// Mitsubishi GX Works2 project: B02_UDE 20260304_0   PLC: Q03UDE

PROGRAM 00  // Prog切替
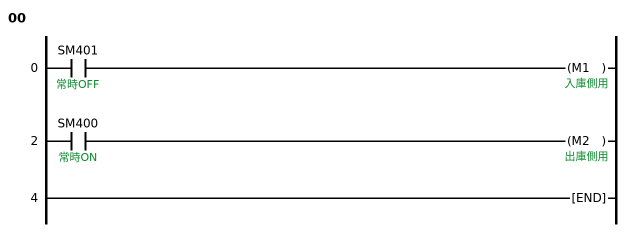
0     LD      SM401  ; 常時OFF
      OUT     M1  ; 入庫側用
2     LD      SM400  ; 常時ON
      OUT     M2  ; 出庫側用
4     END
END_PROGRAM

PROGRAM 01  // IO入力
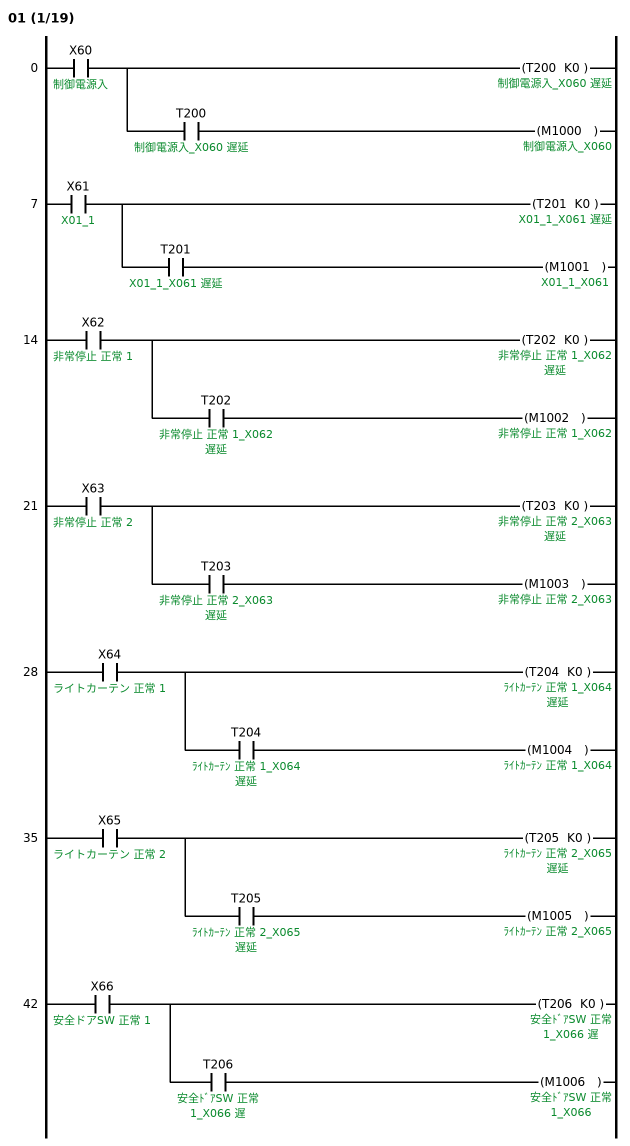
0     LD      X60  ; 制御電源入
      OUT     T200 K0  ; 制御電源入_X060 遅延
      AND     T200  ; 制御電源入_X060 遅延
      OUT     M1000  ; 制御電源入_X060
7     LD      X61  ; X01_1
      OUT     T201 K0  ; X01_1_X061 遅延
      AND     T201  ; X01_1_X061 遅延
      OUT     M1001  ; X01_1_X061
14    LD      X62  ; 非常停止 正常 1
      OUT     T202 K0  ; 非常停止 正常 1_X062 遅延
      AND     T202  ; 非常停止 正常 1_X062 遅延
      OUT     M1002  ; 非常停止 正常 1_X062
21    LD      X63  ; 非常停止 正常 2
      OUT     T203 K0  ; 非常停止 正常 2_X063 遅延
      AND     T203  ; 非常停止 正常 2_X063 遅延
      OUT     M1003  ; 非常停止 正常 2_X063
28    LD      X64  ; ライトカーテン 正常 1
      OUT     T204 K0  ; ﾗｲﾄｶｰﾃﾝ 正常 1_X064 遅延
      AND     T204  ; ﾗｲﾄｶｰﾃﾝ 正常 1_X064 遅延
      OUT     M1004  ; ﾗｲﾄｶｰﾃﾝ 正常 1_X064
35    LD      X65  ; ライトカーテン 正常 2
      OUT     T205 K0  ; ﾗｲﾄｶｰﾃﾝ 正常 2_X065 遅延
      AND     T205  ; ﾗｲﾄｶｰﾃﾝ 正常 2_X065 遅延
      OUT     M1005  ; ﾗｲﾄｶｰﾃﾝ 正常 2_X065
42    LD      X66  ; 安全ドアSW 正常 1
      OUT     T206 K0  ; 安全ﾄﾞｱSW 正常 1_X066 遅
      AND     T206  ; 安全ﾄﾞｱSW 正常 1_X066 遅
      OUT     M1006  ; 安全ﾄﾞｱSW 正常 1_X066
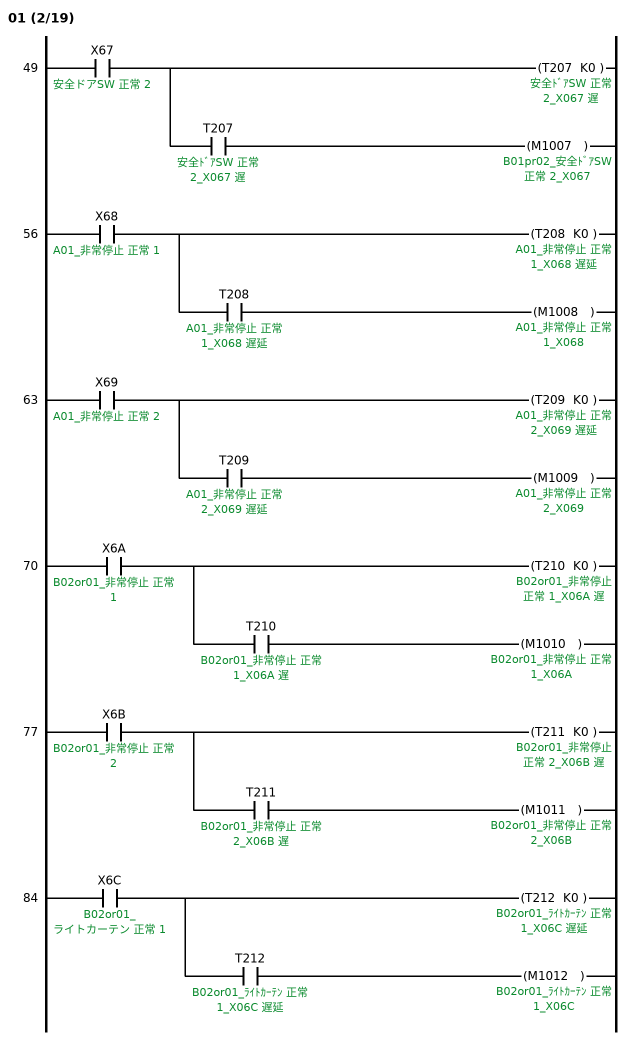
49    LD      X67  ; 安全ドアSW 正常 2
      OUT     T207 K0  ; 安全ﾄﾞｱSW 正常 2_X067 遅
      AND     T207  ; 安全ﾄﾞｱSW 正常 2_X067 遅
      OUT     M1007  ; B01pr02_安全ﾄﾞｱSW 正常 2_X067
56    LD      X68  ; A01_非常停止 正常 1
      OUT     T208 K0  ; A01_非常停止 正常 1_X068 遅延
      AND     T208  ; A01_非常停止 正常 1_X068 遅延
      OUT     M1008  ; A01_非常停止 正常 1_X068
63    LD      X69  ; A01_非常停止 正常 2
      OUT     T209 K0  ; A01_非常停止 正常 2_X069 遅延
      AND     T209  ; A01_非常停止 正常 2_X069 遅延
      OUT     M1009  ; A01_非常停止 正常 2_X069
70    LD      X6A  ; B02or01_非常停止 正常 1
      OUT     T210 K0  ; B02or01_非常停止 正常 1_X06A 遅
      AND     T210  ; B02or01_非常停止 正常 1_X06A 遅
      OUT     M1010  ; B02or01_非常停止 正常 1_X06A
77    LD      X6B  ; B02or01_非常停止 正常 2
      OUT     T211 K0  ; B02or01_非常停止 正常 2_X06B 遅
      AND     T211  ; B02or01_非常停止 正常 2_X06B 遅
      OUT     M1011  ; B02or01_非常停止 正常 2_X06B
84    LD      X6C  ; B02or01_ライトカーテン 正常 1
      OUT     T212 K0  ; B02or01_ﾗｲﾄｶｰﾃﾝ 正常 1_X06C 遅延
      AND     T212  ; B02or01_ﾗｲﾄｶｰﾃﾝ 正常 1_X06C 遅延
      OUT     M1012  ; B02or01_ﾗｲﾄｶｰﾃﾝ 正常 1_X06C
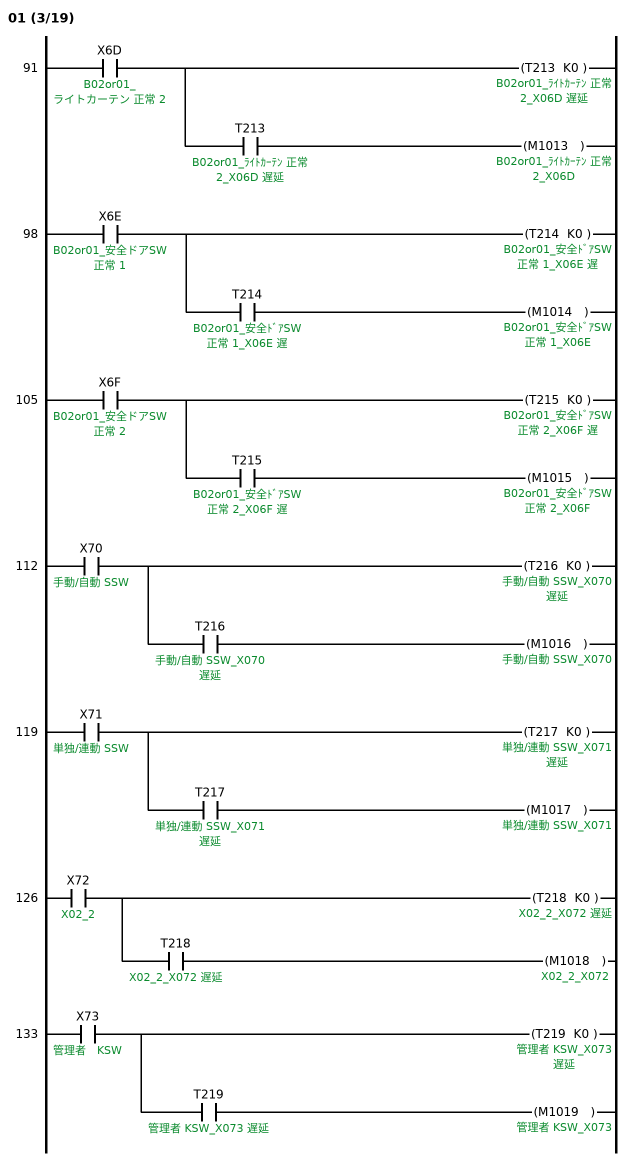
91    LD      X6D  ; B02or01_ライトカーテン 正常 2
      OUT     T213 K0  ; B02or01_ﾗｲﾄｶｰﾃﾝ 正常 2_X06D 遅延
      AND     T213  ; B02or01_ﾗｲﾄｶｰﾃﾝ 正常 2_X06D 遅延
      OUT     M1013  ; B02or01_ﾗｲﾄｶｰﾃﾝ 正常 2_X06D
98    LD      X6E  ; B02or01_安全ドアSW 正常 1
      OUT     T214 K0  ; B02or01_安全ﾄﾞｱSW 正常 1_X06E 遅
      AND     T214  ; B02or01_安全ﾄﾞｱSW 正常 1_X06E 遅
      OUT     M1014  ; B02or01_安全ﾄﾞｱSW 正常 1_X06E
105   LD      X6F  ; B02or01_安全ドアSW 正常 2
      OUT     T215 K0  ; B02or01_安全ﾄﾞｱSW 正常 2_X06F 遅
      AND     T215  ; B02or01_安全ﾄﾞｱSW 正常 2_X06F 遅
      OUT     M1015  ; B02or01_安全ﾄﾞｱSW 正常 2_X06F
112   LD      X70  ; 手動/自動 SSW
      OUT     T216 K0  ; 手動/自動 SSW_X070 遅延
      AND     T216  ; 手動/自動 SSW_X070 遅延
      OUT     M1016  ; 手動/自動 SSW_X070
119   LD      X71  ; 単独/連動 SSW
      OUT     T217 K0  ; 単独/連動 SSW_X071 遅延
      AND     T217  ; 単独/連動 SSW_X071 遅延
      OUT     M1017  ; 単独/連動 SSW_X071
126   LD      X72  ; X02_2
      OUT     T218 K0  ; X02_2_X072 遅延
      AND     T218  ; X02_2_X072 遅延
      OUT     M1018  ; X02_2_X072
133   LD      X73  ; 管理者　KSW
      OUT     T219 K0  ; 管理者 KSW_X073 遅延
      AND     T219  ; 管理者 KSW_X073 遅延
      OUT     M1019  ; 管理者 KSW_X073
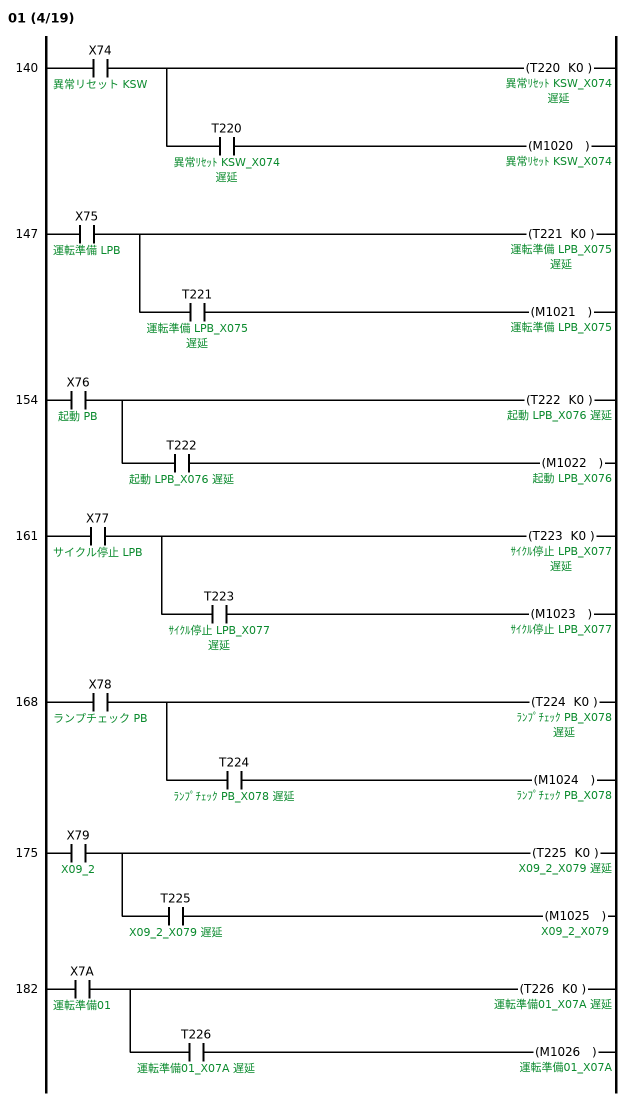
140   LD      X74  ; 異常リセット KSW
      OUT     T220 K0  ; 異常ﾘｾｯﾄ KSW_X074 遅延
      AND     T220  ; 異常ﾘｾｯﾄ KSW_X074 遅延
      OUT     M1020  ; 異常ﾘｾｯﾄ KSW_X074
147   LD      X75  ; 運転準備 LPB
      OUT     T221 K0  ; 運転準備 LPB_X075 遅延
      AND     T221  ; 運転準備 LPB_X075 遅延
      OUT     M1021  ; 運転準備 LPB_X075
154   LD      X76  ; 起動 PB
      OUT     T222 K0  ; 起動 LPB_X076 遅延
      AND     T222  ; 起動 LPB_X076 遅延
      OUT     M1022  ; 起動 LPB_X076
161   LD      X77  ; サイクル停止 LPB
      OUT     T223 K0  ; ｻｲｸﾙ停止 LPB_X077 遅延
      AND     T223  ; ｻｲｸﾙ停止 LPB_X077 遅延
      OUT     M1023  ; ｻｲｸﾙ停止 LPB_X077
168   LD      X78  ; ランプチェック PB
      OUT     T224 K0  ; ﾗﾝﾌﾟﾁｪｯｸ PB_X078 遅延
      AND     T224  ; ﾗﾝﾌﾟﾁｪｯｸ PB_X078 遅延
      OUT     M1024  ; ﾗﾝﾌﾟﾁｪｯｸ PB_X078
175   LD      X79  ; X09_2
      OUT     T225 K0  ; X09_2_X079 遅延
      AND     T225  ; X09_2_X079 遅延
      OUT     M1025  ; X09_2_X079
182   LD      X7A  ; 運転準備01
      OUT     T226 K0  ; 運転準備01_X07A 遅延
      AND     T226  ; 運転準備01_X07A 遅延
      OUT     M1026  ; 運転準備01_X07A
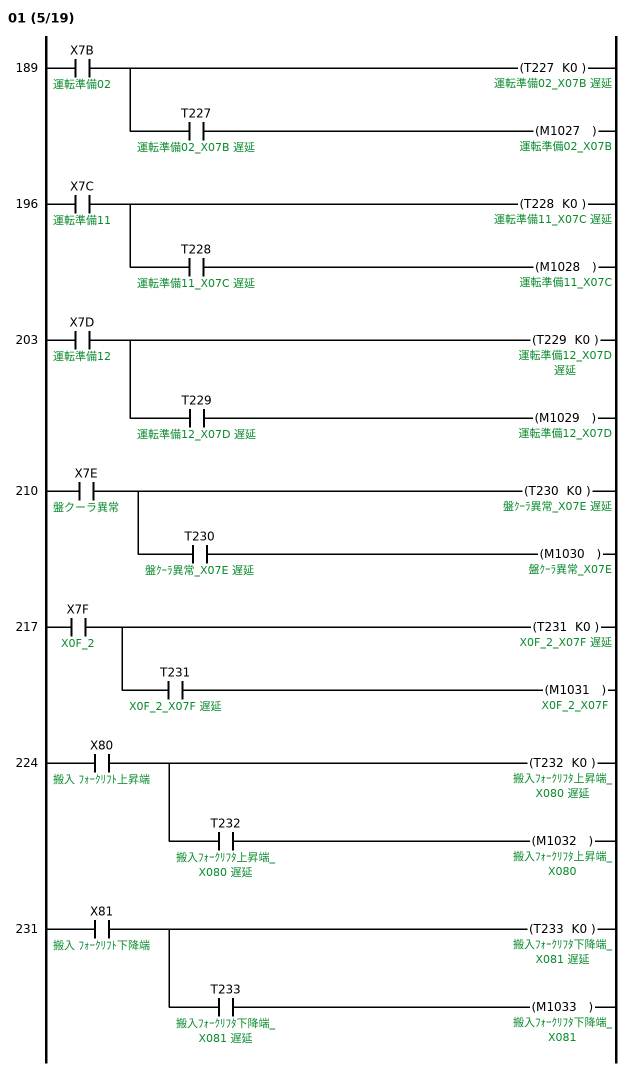
189   LD      X7B  ; 運転準備02
      OUT     T227 K0  ; 運転準備02_X07B 遅延
      AND     T227  ; 運転準備02_X07B 遅延
      OUT     M1027  ; 運転準備02_X07B
196   LD      X7C  ; 運転準備11
      OUT     T228 K0  ; 運転準備11_X07C 遅延
      AND     T228  ; 運転準備11_X07C 遅延
      OUT     M1028  ; 運転準備11_X07C
203   LD      X7D  ; 運転準備12
      OUT     T229 K0  ; 運転準備12_X07D 遅延
      AND     T229  ; 運転準備12_X07D 遅延
      OUT     M1029  ; 運転準備12_X07D
210   LD      X7E  ; 盤クーラ異常
      OUT     T230 K0  ; 盤ｸｰﾗ異常_X07E 遅延
      AND     T230  ; 盤ｸｰﾗ異常_X07E 遅延
      OUT     M1030  ; 盤ｸｰﾗ異常_X07E
217   LD      X7F  ; X0F_2
      OUT     T231 K0  ; X0F_2_X07F 遅延
      AND     T231  ; X0F_2_X07F 遅延
      OUT     M1031  ; X0F_2_X07F
224   LD      X80  ; 搬入 ﾌｫｰｸﾘﾌﾄ上昇端
      OUT     T232 K0  ; 搬入ﾌｫｰｸﾘﾌﾀ上昇端_X080 遅延
      AND     T232  ; 搬入ﾌｫｰｸﾘﾌﾀ上昇端_X080 遅延
      OUT     M1032  ; 搬入ﾌｫｰｸﾘﾌﾀ上昇端_X080
231   LD      X81  ; 搬入 ﾌｫｰｸﾘﾌﾄ下降端
      OUT     T233 K0  ; 搬入ﾌｫｰｸﾘﾌﾀ下降端_X081 遅延
      AND     T233  ; 搬入ﾌｫｰｸﾘﾌﾀ下降端_X081 遅延
      OUT     M1033  ; 搬入ﾌｫｰｸﾘﾌﾀ下降端_X081
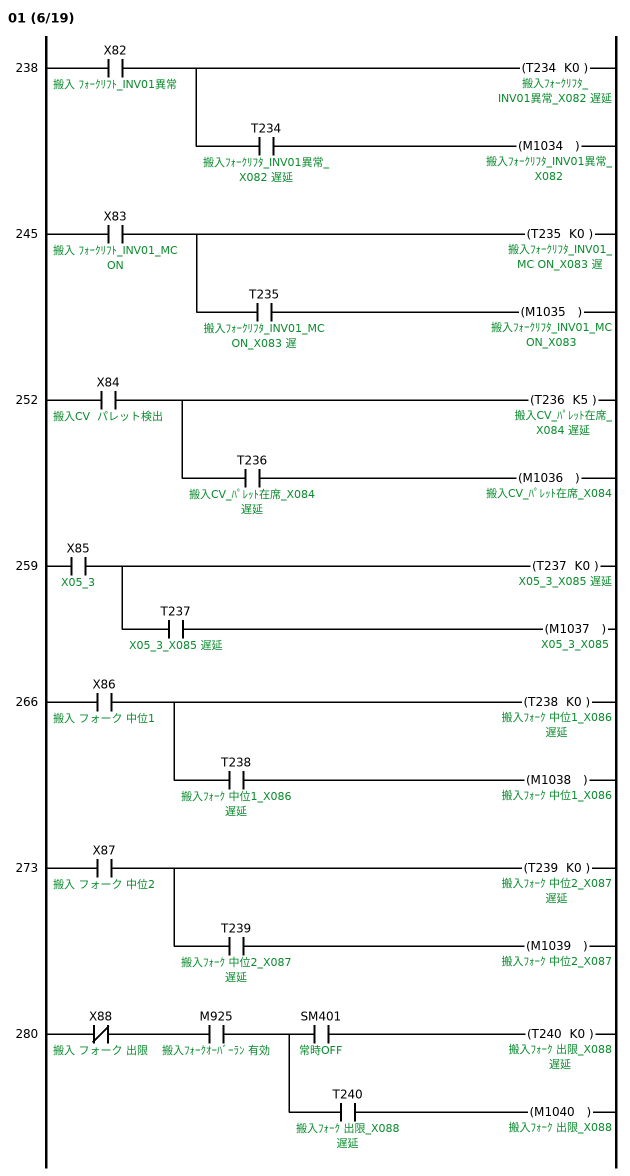
238   LD      X82  ; 搬入 ﾌｫｰｸﾘﾌﾄ_INV01異常
      OUT     T234 K0  ; 搬入ﾌｫｰｸﾘﾌﾀ_INV01異常_X082 遅延
      AND     T234  ; 搬入ﾌｫｰｸﾘﾌﾀ_INV01異常_X082 遅延
      OUT     M1034  ; 搬入ﾌｫｰｸﾘﾌﾀ_INV01異常_X082
245   LD      X83  ; 搬入 ﾌｫｰｸﾘﾌﾄ_INV01_MC ON
      OUT     T235 K0  ; 搬入ﾌｫｰｸﾘﾌﾀ_INV01_MC ON_X083 遅
      AND     T235  ; 搬入ﾌｫｰｸﾘﾌﾀ_INV01_MC ON_X083 遅
      OUT     M1035  ; 搬入ﾌｫｰｸﾘﾌﾀ_INV01_MC ON_X083
252   LD      X84  ; 搬入CV  パレット検出
      OUT     T236 K5  ; 搬入CV_ﾊﾟﾚｯﾄ在席_X084 遅延
      AND     T236  ; 搬入CV_ﾊﾟﾚｯﾄ在席_X084 遅延
      OUT     M1036  ; 搬入CV_ﾊﾟﾚｯﾄ在席_X084
259   LD      X85  ; X05_3
      OUT     T237 K0  ; X05_3_X085 遅延
      AND     T237  ; X05_3_X085 遅延
      OUT     M1037  ; X05_3_X085
266   LD      X86  ; 搬入 フォーク 中位1
      OUT     T238 K0  ; 搬入ﾌｫｰｸ 中位1_X086 遅延
      AND     T238  ; 搬入ﾌｫｰｸ 中位1_X086 遅延
      OUT     M1038  ; 搬入ﾌｫｰｸ 中位1_X086
273   LD      X87  ; 搬入 フォーク 中位2
      OUT     T239 K0  ; 搬入ﾌｫｰｸ 中位2_X087 遅延
      AND     T239  ; 搬入ﾌｫｰｸ 中位2_X087 遅延
      OUT     M1039  ; 搬入ﾌｫｰｸ 中位2_X087
280   LDI     X88  ; 搬入 フォーク 出限
      AND     M925  ; 搬入ﾌｫｰｸｵｰﾊﾞｰﾗﾝ 有効
      MPS
      AND     SM401  ; 常時OFF
      OUT     T240 K0  ; 搬入ﾌｫｰｸ 出限_X088 遅延
      MPP
      AND     T240  ; 搬入ﾌｫｰｸ 出限_X088 遅延
      OUT     M1040  ; 搬入ﾌｫｰｸ 出限_X088
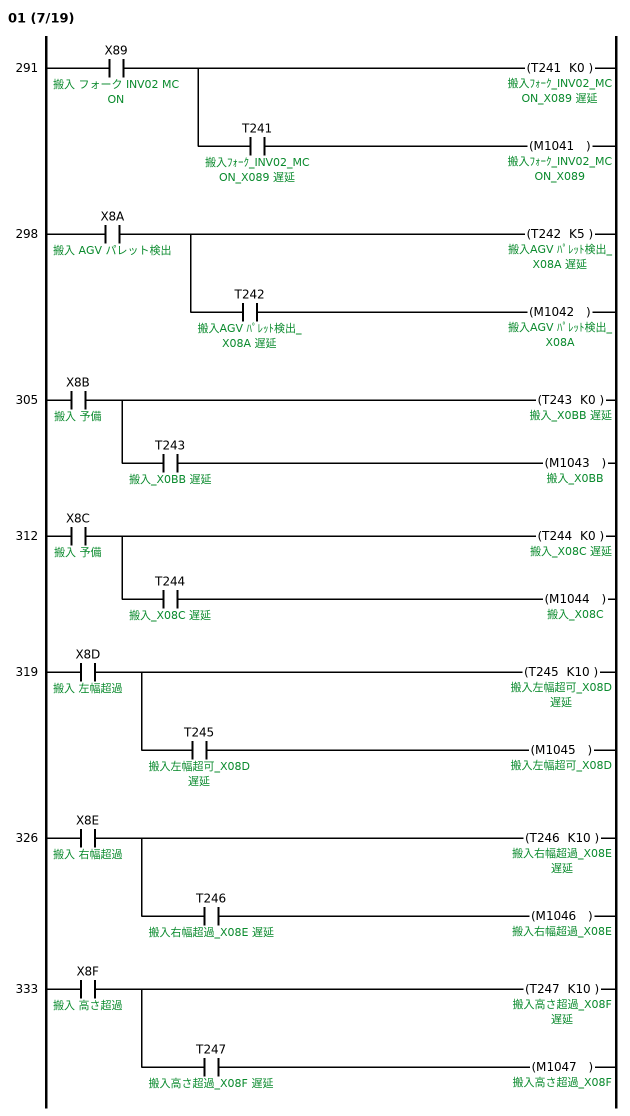
291   LD      X89  ; 搬入 フォーク INV02 MC ON
      OUT     T241 K0  ; 搬入ﾌｫｰｸ_INV02_MC ON_X089 遅延
      AND     T241  ; 搬入ﾌｫｰｸ_INV02_MC ON_X089 遅延
      OUT     M1041  ; 搬入ﾌｫｰｸ_INV02_MC ON_X089
298   LD      X8A  ; 搬入 AGV パレット検出
      OUT     T242 K5  ; 搬入AGV ﾊﾟﾚｯﾄ検出_X08A 遅延
      AND     T242  ; 搬入AGV ﾊﾟﾚｯﾄ検出_X08A 遅延
      OUT     M1042  ; 搬入AGV ﾊﾟﾚｯﾄ検出_X08A
305   LD      X8B  ; 搬入 予備
      OUT     T243 K0  ; 搬入_X0BB 遅延
      AND     T243  ; 搬入_X0BB 遅延
      OUT     M1043  ; 搬入_X0BB
312   LD      X8C  ; 搬入 予備
      OUT     T244 K0  ; 搬入_X08C 遅延
      AND     T244  ; 搬入_X08C 遅延
      OUT     M1044  ; 搬入_X08C
319   LD      X8D  ; 搬入 左幅超過
      OUT     T245 K10  ; 搬入左幅超可_X08D 遅延
      AND     T245  ; 搬入左幅超可_X08D 遅延
      OUT     M1045  ; 搬入左幅超可_X08D
326   LD      X8E  ; 搬入 右幅超過
      OUT     T246 K10  ; 搬入右幅超過_X08E 遅延
      AND     T246  ; 搬入右幅超過_X08E 遅延
      OUT     M1046  ; 搬入右幅超過_X08E
333   LD      X8F  ; 搬入 高さ超過
      OUT     T247 K10  ; 搬入高さ超過_X08F 遅延
      AND     T247  ; 搬入高さ超過_X08F 遅延
      OUT     M1047  ; 搬入高さ超過_X08F
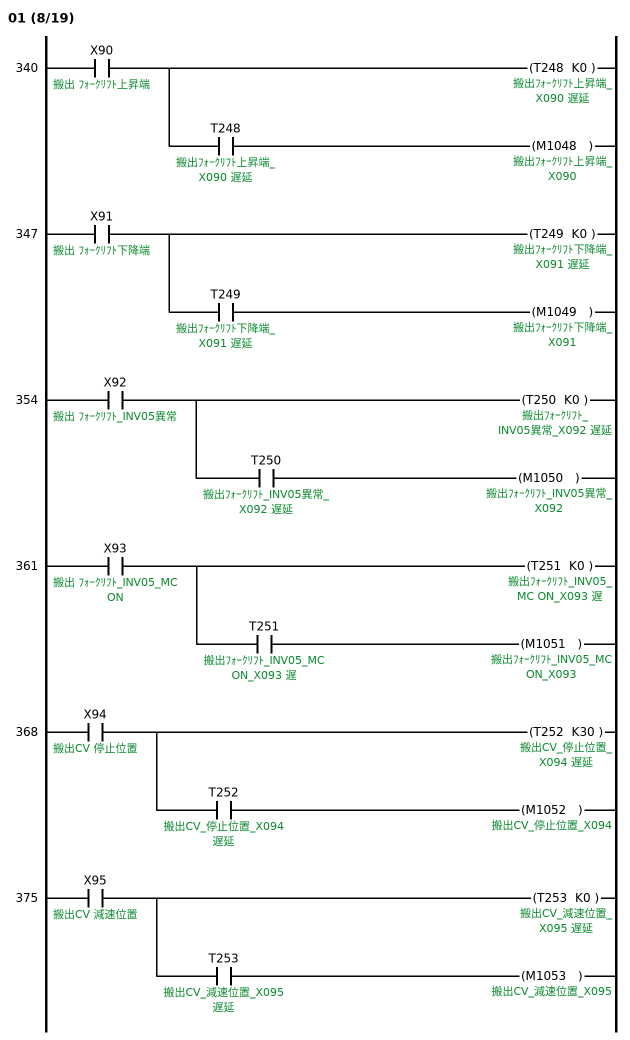
340   LD      X90  ; 搬出 ﾌｫｰｸﾘﾌﾄ上昇端
      OUT     T248 K0  ; 搬出ﾌｫｰｸﾘﾌﾄ上昇端_X090 遅延
      AND     T248  ; 搬出ﾌｫｰｸﾘﾌﾄ上昇端_X090 遅延
      OUT     M1048  ; 搬出ﾌｫｰｸﾘﾌﾄ上昇端_X090
347   LD      X91  ; 搬出 ﾌｫｰｸﾘﾌﾄ下降端
      OUT     T249 K0  ; 搬出ﾌｫｰｸﾘﾌﾄ下降端_X091 遅延
      AND     T249  ; 搬出ﾌｫｰｸﾘﾌﾄ下降端_X091 遅延
      OUT     M1049  ; 搬出ﾌｫｰｸﾘﾌﾄ下降端_X091
354   LD      X92  ; 搬出 ﾌｫｰｸﾘﾌﾄ_INV05異常
      OUT     T250 K0  ; 搬出ﾌｫｰｸﾘﾌﾄ_INV05異常_X092 遅延
      AND     T250  ; 搬出ﾌｫｰｸﾘﾌﾄ_INV05異常_X092 遅延
      OUT     M1050  ; 搬出ﾌｫｰｸﾘﾌﾄ_INV05異常_X092
361   LD      X93  ; 搬出 ﾌｫｰｸﾘﾌﾄ_INV05_MC ON
      OUT     T251 K0  ; 搬出ﾌｫｰｸﾘﾌﾄ_INV05_MC ON_X093 遅
      AND     T251  ; 搬出ﾌｫｰｸﾘﾌﾄ_INV05_MC ON_X093 遅
      OUT     M1051  ; 搬出ﾌｫｰｸﾘﾌﾄ_INV05_MC ON_X093
368   LD      X94  ; 搬出CV 停止位置
      OUT     T252 K30  ; 搬出CV_停止位置_X094 遅延
      AND     T252  ; 搬出CV_停止位置_X094 遅延
      OUT     M1052  ; 搬出CV_停止位置_X094
375   LD      X95  ; 搬出CV 減速位置
      OUT     T253 K0  ; 搬出CV_減速位置_X095 遅延
      AND     T253  ; 搬出CV_減速位置_X095 遅延
      OUT     M1053  ; 搬出CV_減速位置_X095
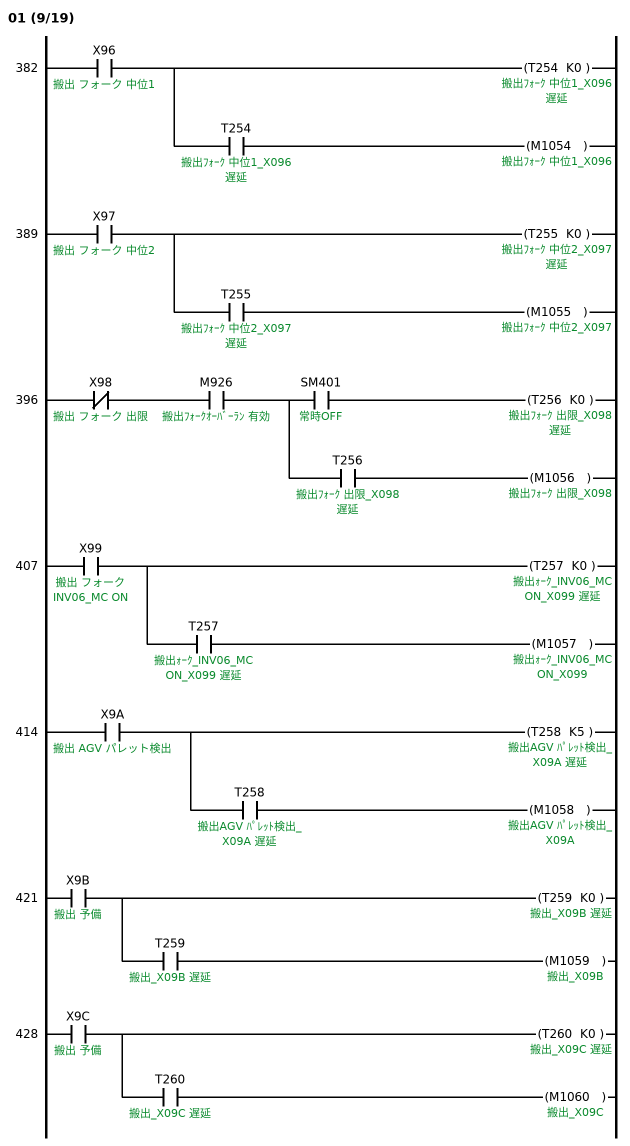
382   LD      X96  ; 搬出 フォーク 中位1
      OUT     T254 K0  ; 搬出ﾌｫｰｸ 中位1_X096 遅延
      AND     T254  ; 搬出ﾌｫｰｸ 中位1_X096 遅延
      OUT     M1054  ; 搬出ﾌｫｰｸ 中位1_X096
389   LD      X97  ; 搬出 フォーク 中位2
      OUT     T255 K0  ; 搬出ﾌｫｰｸ 中位2_X097 遅延
      AND     T255  ; 搬出ﾌｫｰｸ 中位2_X097 遅延
      OUT     M1055  ; 搬出ﾌｫｰｸ 中位2_X097
396   LDI     X98  ; 搬出 フォーク 出限
      AND     M926  ; 搬出ﾌｫｰｸｵｰﾊﾞｰﾗﾝ 有効
      MPS
      AND     SM401  ; 常時OFF
      OUT     T256 K0  ; 搬出ﾌｫｰｸ 出限_X098 遅延
      MPP
      AND     T256  ; 搬出ﾌｫｰｸ 出限_X098 遅延
      OUT     M1056  ; 搬出ﾌｫｰｸ 出限_X098
407   LD      X99  ; 搬出 フォーク INV06_MC ON
      OUT     T257 K0  ; 搬出ｫｰｸ_INV06_MC ON_X099 遅延
      AND     T257  ; 搬出ｫｰｸ_INV06_MC ON_X099 遅延
      OUT     M1057  ; 搬出ｫｰｸ_INV06_MC ON_X099
414   LD      X9A  ; 搬出 AGV パレット検出
      OUT     T258 K5  ; 搬出AGV ﾊﾟﾚｯﾄ検出_X09A 遅延
      AND     T258  ; 搬出AGV ﾊﾟﾚｯﾄ検出_X09A 遅延
      OUT     M1058  ; 搬出AGV ﾊﾟﾚｯﾄ検出_X09A
421   LD      X9B  ; 搬出 予備
      OUT     T259 K0  ; 搬出_X09B 遅延
      AND     T259  ; 搬出_X09B 遅延
      OUT     M1059  ; 搬出_X09B
428   LD      X9C  ; 搬出 予備
      OUT     T260 K0  ; 搬出_X09C 遅延
      AND     T260  ; 搬出_X09C 遅延
      OUT     M1060  ; 搬出_X09C
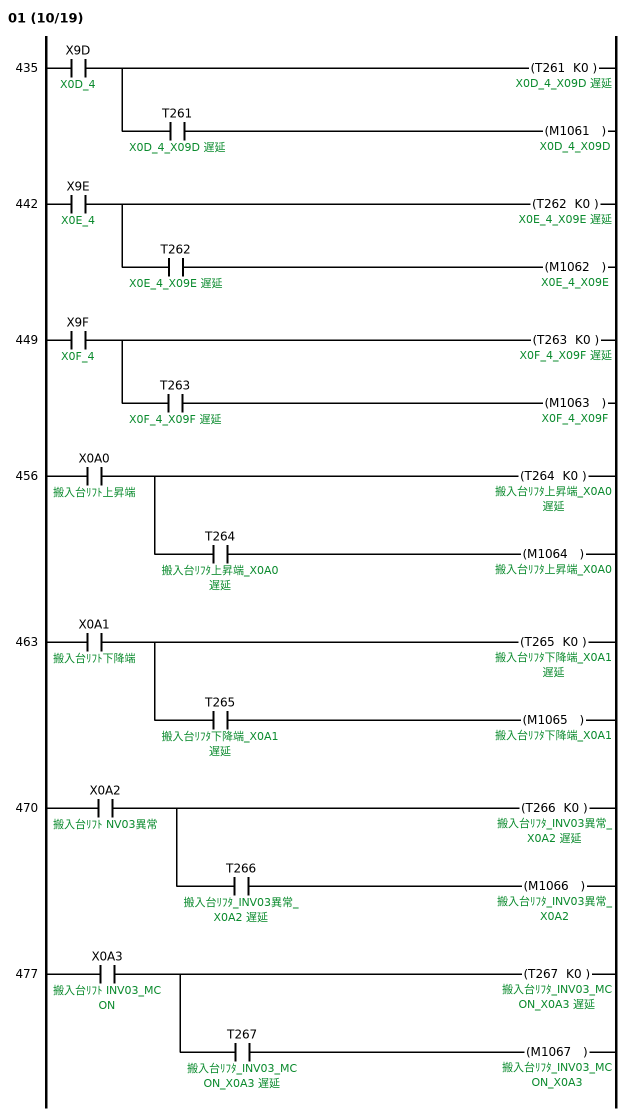
435   LD      X9D  ; X0D_4
      OUT     T261 K0  ; X0D_4_X09D 遅延
      AND     T261  ; X0D_4_X09D 遅延
      OUT     M1061  ; X0D_4_X09D
442   LD      X9E  ; X0E_4
      OUT     T262 K0  ; X0E_4_X09E 遅延
      AND     T262  ; X0E_4_X09E 遅延
      OUT     M1062  ; X0E_4_X09E
449   LD      X9F  ; X0F_4
      OUT     T263 K0  ; X0F_4_X09F 遅延
      AND     T263  ; X0F_4_X09F 遅延
      OUT     M1063  ; X0F_4_X09F
456   LD      X0A0  ; 搬入台ﾘﾌﾄ上昇端
      OUT     T264 K0  ; 搬入台ﾘﾌﾀ上昇端_X0A0 遅延
      AND     T264  ; 搬入台ﾘﾌﾀ上昇端_X0A0 遅延
      OUT     M1064  ; 搬入台ﾘﾌﾀ上昇端_X0A0
463   LD      X0A1  ; 搬入台ﾘﾌﾄ下降端
      OUT     T265 K0  ; 搬入台ﾘﾌﾀ下降端_X0A1 遅延
      AND     T265  ; 搬入台ﾘﾌﾀ下降端_X0A1 遅延
      OUT     M1065  ; 搬入台ﾘﾌﾀ下降端_X0A1
470   LD      X0A2  ; 搬入台ﾘﾌﾄ NV03異常
      OUT     T266 K0  ; 搬入台ﾘﾌﾀ_INV03異常_X0A2 遅延
      AND     T266  ; 搬入台ﾘﾌﾀ_INV03異常_X0A2 遅延
      OUT     M1066  ; 搬入台ﾘﾌﾀ_INV03異常_X0A2
477   LD      X0A3  ; 搬入台ﾘﾌﾄ INV03_MC ON
      OUT     T267 K0  ; 搬入台ﾘﾌﾀ_INV03_MC ON_X0A3 遅延
      AND     T267  ; 搬入台ﾘﾌﾀ_INV03_MC ON_X0A3 遅延
      OUT     M1067  ; 搬入台ﾘﾌﾀ_INV03_MC ON_X0A3
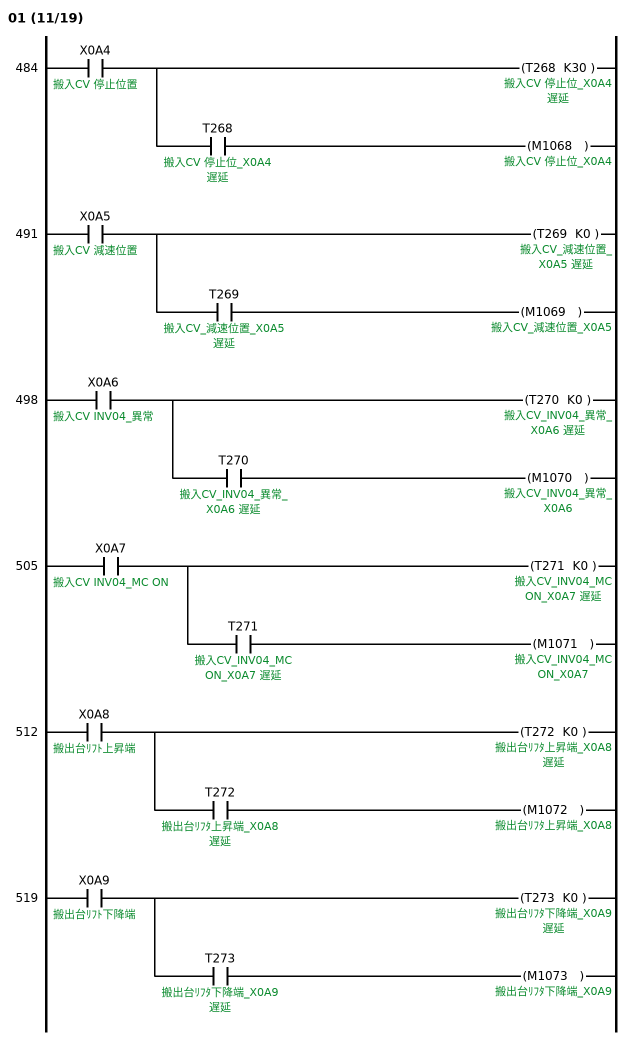
484   LD      X0A4  ; 搬入CV 停止位置
      OUT     T268 K30  ; 搬入CV 停止位_X0A4 遅延
      AND     T268  ; 搬入CV 停止位_X0A4 遅延
      OUT     M1068  ; 搬入CV 停止位_X0A4
491   LD      X0A5  ; 搬入CV 減速位置
      OUT     T269 K0  ; 搬入CV_減速位置_X0A5 遅延
      AND     T269  ; 搬入CV_減速位置_X0A5 遅延
      OUT     M1069  ; 搬入CV_減速位置_X0A5
498   LD      X0A6  ; 搬入CV INV04_異常
      OUT     T270 K0  ; 搬入CV_INV04_異常_X0A6 遅延
      AND     T270  ; 搬入CV_INV04_異常_X0A6 遅延
      OUT     M1070  ; 搬入CV_INV04_異常_X0A6
505   LD      X0A7  ; 搬入CV INV04_MC ON
      OUT     T271 K0  ; 搬入CV_INV04_MC ON_X0A7 遅延
      AND     T271  ; 搬入CV_INV04_MC ON_X0A7 遅延
      OUT     M1071  ; 搬入CV_INV04_MC ON_X0A7
512   LD      X0A8  ; 搬出台ﾘﾌﾄ上昇端
      OUT     T272 K0  ; 搬出台ﾘﾌﾀ上昇端_X0A8 遅延
      AND     T272  ; 搬出台ﾘﾌﾀ上昇端_X0A8 遅延
      OUT     M1072  ; 搬出台ﾘﾌﾀ上昇端_X0A8
519   LD      X0A9  ; 搬出台ﾘﾌﾄ下降端
      OUT     T273 K0  ; 搬出台ﾘﾌﾀ下降端_X0A9 遅延
      AND     T273  ; 搬出台ﾘﾌﾀ下降端_X0A9 遅延
      OUT     M1073  ; 搬出台ﾘﾌﾀ下降端_X0A9
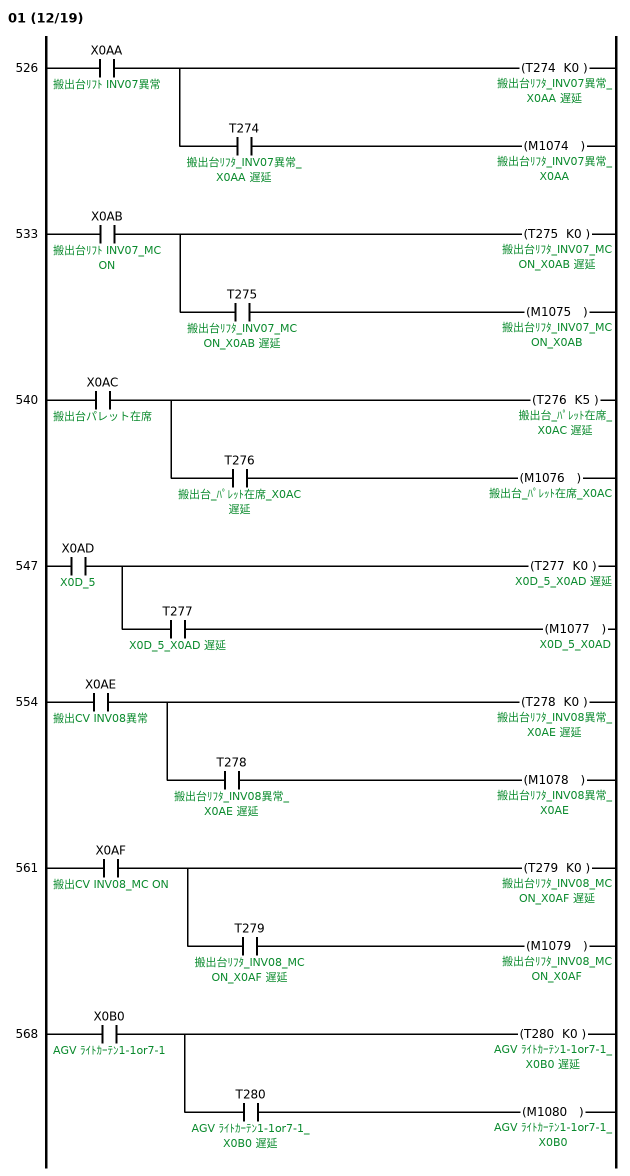
526   LD      X0AA  ; 搬出台ﾘﾌﾄ INV07異常
      OUT     T274 K0  ; 搬出台ﾘﾌﾀ_INV07異常_X0AA 遅延
      AND     T274  ; 搬出台ﾘﾌﾀ_INV07異常_X0AA 遅延
      OUT     M1074  ; 搬出台ﾘﾌﾀ_INV07異常_X0AA
533   LD      X0AB  ; 搬出台ﾘﾌﾄ INV07_MC ON
      OUT     T275 K0  ; 搬出台ﾘﾌﾀ_INV07_MC ON_X0AB 遅延
      AND     T275  ; 搬出台ﾘﾌﾀ_INV07_MC ON_X0AB 遅延
      OUT     M1075  ; 搬出台ﾘﾌﾀ_INV07_MC ON_X0AB
540   LD      X0AC  ; 搬出台パレット在席
      OUT     T276 K5  ; 搬出台_ﾊﾟﾚｯﾄ在席_X0AC 遅延
      AND     T276  ; 搬出台_ﾊﾟﾚｯﾄ在席_X0AC 遅延
      OUT     M1076  ; 搬出台_ﾊﾟﾚｯﾄ在席_X0AC
547   LD      X0AD  ; X0D_5
      OUT     T277 K0  ; X0D_5_X0AD 遅延
      AND     T277  ; X0D_5_X0AD 遅延
      OUT     M1077  ; X0D_5_X0AD
554   LD      X0AE  ; 搬出CV INV08異常
      OUT     T278 K0  ; 搬出台ﾘﾌﾀ_INV08異常_X0AE 遅延
      AND     T278  ; 搬出台ﾘﾌﾀ_INV08異常_X0AE 遅延
      OUT     M1078  ; 搬出台ﾘﾌﾀ_INV08異常_X0AE
561   LD      X0AF  ; 搬出CV INV08_MC ON
      OUT     T279 K0  ; 搬出台ﾘﾌﾀ_INV08_MC ON_X0AF 遅延
      AND     T279  ; 搬出台ﾘﾌﾀ_INV08_MC ON_X0AF 遅延
      OUT     M1079  ; 搬出台ﾘﾌﾀ_INV08_MC ON_X0AF
568   LD      X0B0  ; AGV ﾗｲﾄｶｰﾃﾝ1-1or7-1
      OUT     T280 K0  ; AGV ﾗｲﾄｶｰﾃﾝ1-1or7-1_X0B0 遅延
      AND     T280  ; AGV ﾗｲﾄｶｰﾃﾝ1-1or7-1_X0B0 遅延
      OUT     M1080  ; AGV ﾗｲﾄｶｰﾃﾝ1-1or7-1_X0B0
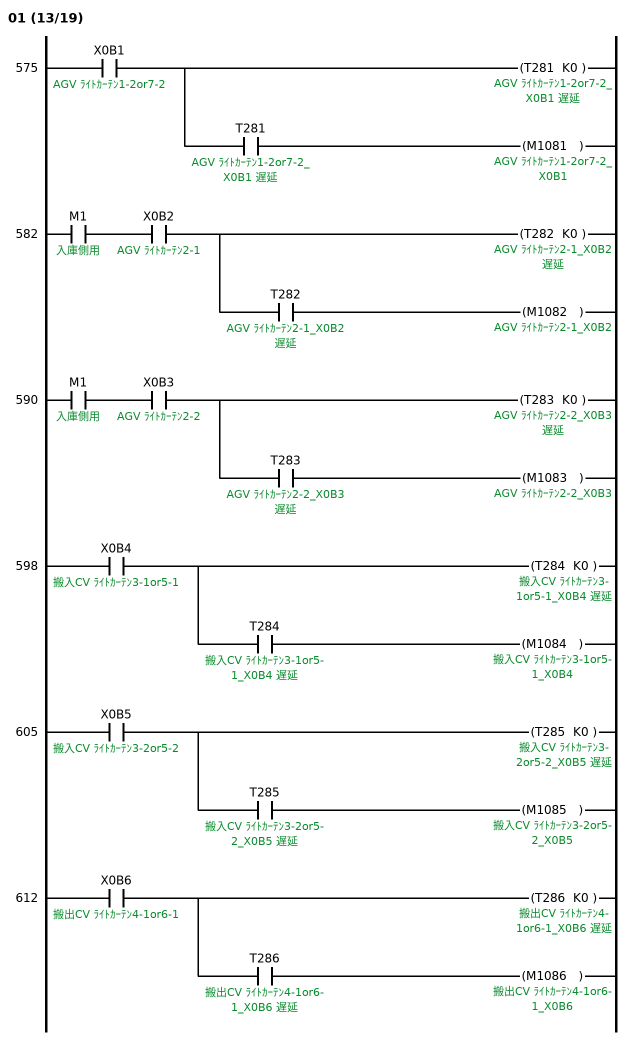
575   LD      X0B1  ; AGV ﾗｲﾄｶｰﾃﾝ1-2or7-2
      OUT     T281 K0  ; AGV ﾗｲﾄｶｰﾃﾝ1-2or7-2_X0B1 遅延
      AND     T281  ; AGV ﾗｲﾄｶｰﾃﾝ1-2or7-2_X0B1 遅延
      OUT     M1081  ; AGV ﾗｲﾄｶｰﾃﾝ1-2or7-2_X0B1
582   LD      M1  ; 入庫側用
      AND     X0B2  ; AGV ﾗｲﾄｶｰﾃﾝ2-1
      OUT     T282 K0  ; AGV ﾗｲﾄｶｰﾃﾝ2-1_X0B2 遅延
      AND     T282  ; AGV ﾗｲﾄｶｰﾃﾝ2-1_X0B2 遅延
      OUT     M1082  ; AGV ﾗｲﾄｶｰﾃﾝ2-1_X0B2
590   LD      M1  ; 入庫側用
      AND     X0B3  ; AGV ﾗｲﾄｶｰﾃﾝ2-2
      OUT     T283 K0  ; AGV ﾗｲﾄｶｰﾃﾝ2-2_X0B3 遅延
      AND     T283  ; AGV ﾗｲﾄｶｰﾃﾝ2-2_X0B3 遅延
      OUT     M1083  ; AGV ﾗｲﾄｶｰﾃﾝ2-2_X0B3
598   LD      X0B4  ; 搬入CV ﾗｲﾄｶｰﾃﾝ3-1or5-1
      OUT     T284 K0  ; 搬入CV ﾗｲﾄｶｰﾃﾝ3-1or5-1_X0B4 遅延
      AND     T284  ; 搬入CV ﾗｲﾄｶｰﾃﾝ3-1or5-1_X0B4 遅延
      OUT     M1084  ; 搬入CV ﾗｲﾄｶｰﾃﾝ3-1or5-1_X0B4
605   LD      X0B5  ; 搬入CV ﾗｲﾄｶｰﾃﾝ3-2or5-2
      OUT     T285 K0  ; 搬入CV ﾗｲﾄｶｰﾃﾝ3-2or5-2_X0B5 遅延
      AND     T285  ; 搬入CV ﾗｲﾄｶｰﾃﾝ3-2or5-2_X0B5 遅延
      OUT     M1085  ; 搬入CV ﾗｲﾄｶｰﾃﾝ3-2or5-2_X0B5
612   LD      X0B6  ; 搬出CV ﾗｲﾄｶｰﾃﾝ4-1or6-1
      OUT     T286 K0  ; 搬出CV ﾗｲﾄｶｰﾃﾝ4-1or6-1_X0B6 遅延
      AND     T286  ; 搬出CV ﾗｲﾄｶｰﾃﾝ4-1or6-1_X0B6 遅延
      OUT     M1086  ; 搬出CV ﾗｲﾄｶｰﾃﾝ4-1or6-1_X0B6
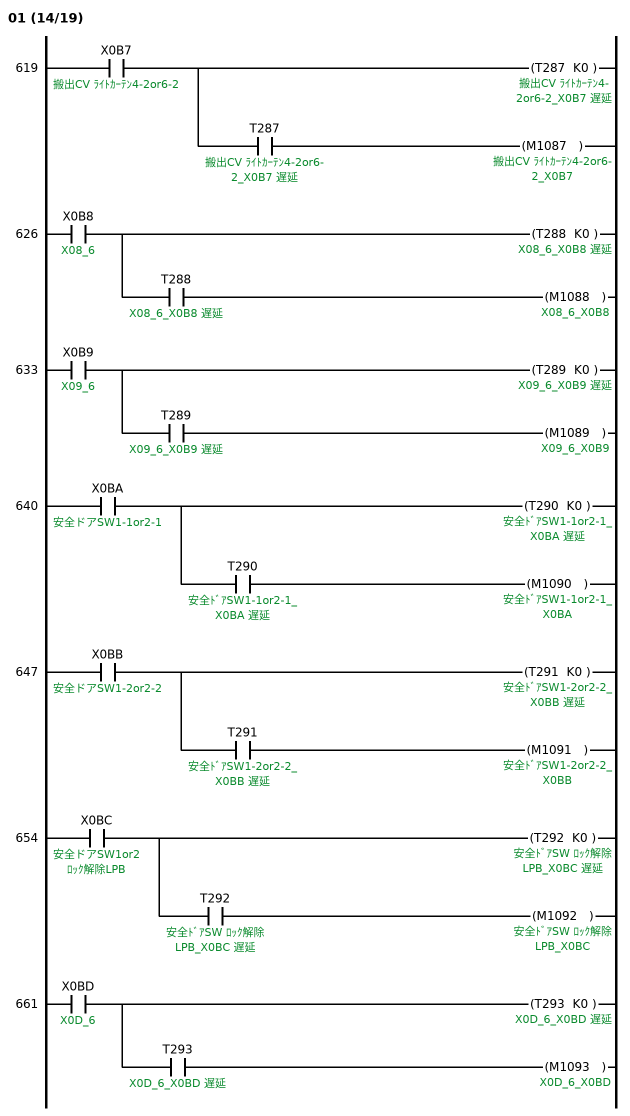
619   LD      X0B7  ; 搬出CV ﾗｲﾄｶｰﾃﾝ4-2or6-2
      OUT     T287 K0  ; 搬出CV ﾗｲﾄｶｰﾃﾝ4-2or6-2_X0B7 遅延
      AND     T287  ; 搬出CV ﾗｲﾄｶｰﾃﾝ4-2or6-2_X0B7 遅延
      OUT     M1087  ; 搬出CV ﾗｲﾄｶｰﾃﾝ4-2or6-2_X0B7
626   LD      X0B8  ; X08_6
      OUT     T288 K0  ; X08_6_X0B8 遅延
      AND     T288  ; X08_6_X0B8 遅延
      OUT     M1088  ; X08_6_X0B8
633   LD      X0B9  ; X09_6
      OUT     T289 K0  ; X09_6_X0B9 遅延
      AND     T289  ; X09_6_X0B9 遅延
      OUT     M1089  ; X09_6_X0B9
640   LD      X0BA  ; 安全ドアSW1-1or2-1
      OUT     T290 K0  ; 安全ﾄﾞｱSW1-1or2-1_X0BA 遅延
      AND     T290  ; 安全ﾄﾞｱSW1-1or2-1_X0BA 遅延
      OUT     M1090  ; 安全ﾄﾞｱSW1-1or2-1_X0BA
647   LD      X0BB  ; 安全ドアSW1-2or2-2
      OUT     T291 K0  ; 安全ﾄﾞｱSW1-2or2-2_X0BB 遅延
      AND     T291  ; 安全ﾄﾞｱSW1-2or2-2_X0BB 遅延
      OUT     M1091  ; 安全ﾄﾞｱSW1-2or2-2_X0BB
654   LD      X0BC  ; 安全ドアSW1or2 ﾛｯｸ解除LPB
      OUT     T292 K0  ; 安全ﾄﾞｱSW ﾛｯｸ解除 LPB_X0BC 遅延
      AND     T292  ; 安全ﾄﾞｱSW ﾛｯｸ解除 LPB_X0BC 遅延
      OUT     M1092  ; 安全ﾄﾞｱSW ﾛｯｸ解除 LPB_X0BC
661   LD      X0BD  ; X0D_6
      OUT     T293 K0  ; X0D_6_X0BD 遅延
      AND     T293  ; X0D_6_X0BD 遅延
      OUT     M1093  ; X0D_6_X0BD
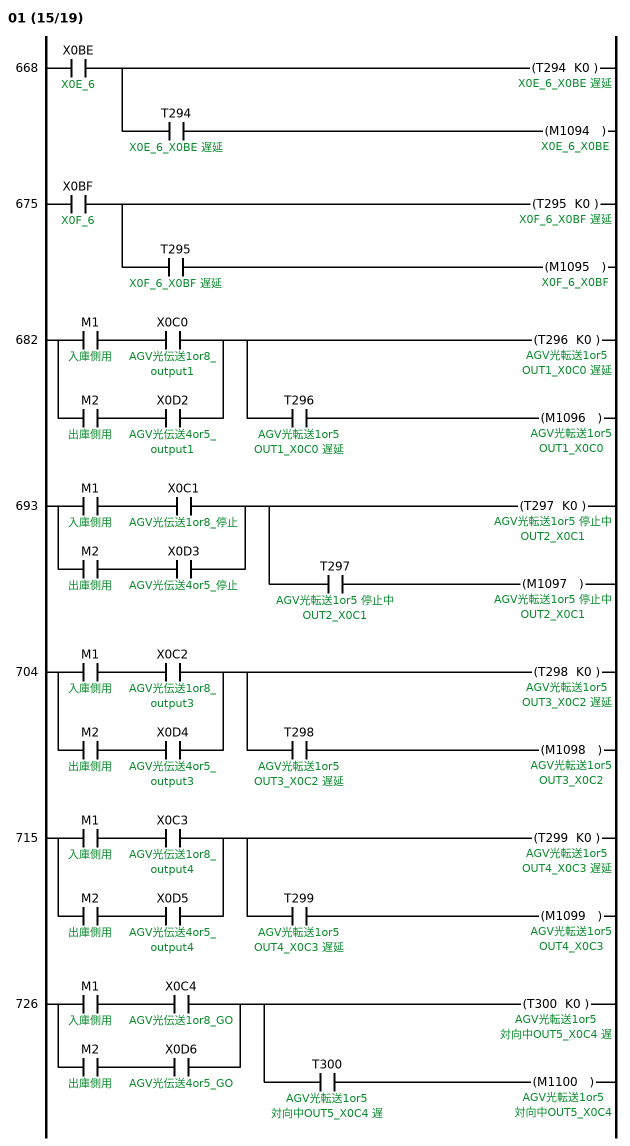
668   LD      X0BE  ; X0E_6
      OUT     T294 K0  ; X0E_6_X0BE 遅延
      AND     T294  ; X0E_6_X0BE 遅延
      OUT     M1094  ; X0E_6_X0BE
675   LD      X0BF  ; X0F_6
      OUT     T295 K0  ; X0F_6_X0BF 遅延
      AND     T295  ; X0F_6_X0BF 遅延
      OUT     M1095  ; X0F_6_X0BF
682   LD      M1  ; 入庫側用
      AND     X0C0  ; AGV光伝送1or8_output1
      LD      M2  ; 出庫側用
      AND     X0D2  ; AGV光伝送4or5_output1
      ORB
      OUT     T296 K0  ; AGV光転送1or5 OUT1_X0C0 遅延
      AND     T296  ; AGV光転送1or5 OUT1_X0C0 遅延
      OUT     M1096  ; AGV光転送1or5 OUT1_X0C0
693   LD      M1  ; 入庫側用
      AND     X0C1  ; AGV光伝送1or8_停止
      LD      M2  ; 出庫側用
      AND     X0D3  ; AGV光伝送4or5_停止
      ORB
      OUT     T297 K0  ; AGV光転送1or5 停止中 OUT2_X0C1
      AND     T297  ; AGV光転送1or5 停止中 OUT2_X0C1
      OUT     M1097  ; AGV光転送1or5 停止中 OUT2_X0C1
704   LD      M1  ; 入庫側用
      AND     X0C2  ; AGV光伝送1or8_output3
      LD      M2  ; 出庫側用
      AND     X0D4  ; AGV光伝送4or5_output3
      ORB
      OUT     T298 K0  ; AGV光転送1or5 OUT3_X0C2 遅延
      AND     T298  ; AGV光転送1or5 OUT3_X0C2 遅延
      OUT     M1098  ; AGV光転送1or5 OUT3_X0C2
715   LD      M1  ; 入庫側用
      AND     X0C3  ; AGV光伝送1or8_output4
      LD      M2  ; 出庫側用
      AND     X0D5  ; AGV光伝送4or5_output4
      ORB
      OUT     T299 K0  ; AGV光転送1or5 OUT4_X0C3 遅延
      AND     T299  ; AGV光転送1or5 OUT4_X0C3 遅延
      OUT     M1099  ; AGV光転送1or5 OUT4_X0C3
726   LD      M1  ; 入庫側用
      AND     X0C4  ; AGV光伝送1or8_GO
      LD      M2  ; 出庫側用
      AND     X0D6  ; AGV光伝送4or5_GO
      ORB
      OUT     T300 K0  ; AGV光転送1or5 対向中OUT5_X0C4 遅
      AND     T300  ; AGV光転送1or5 対向中OUT5_X0C4 遅
      OUT     M1100  ; AGV光転送1or5 対向中OUT5_X0C4
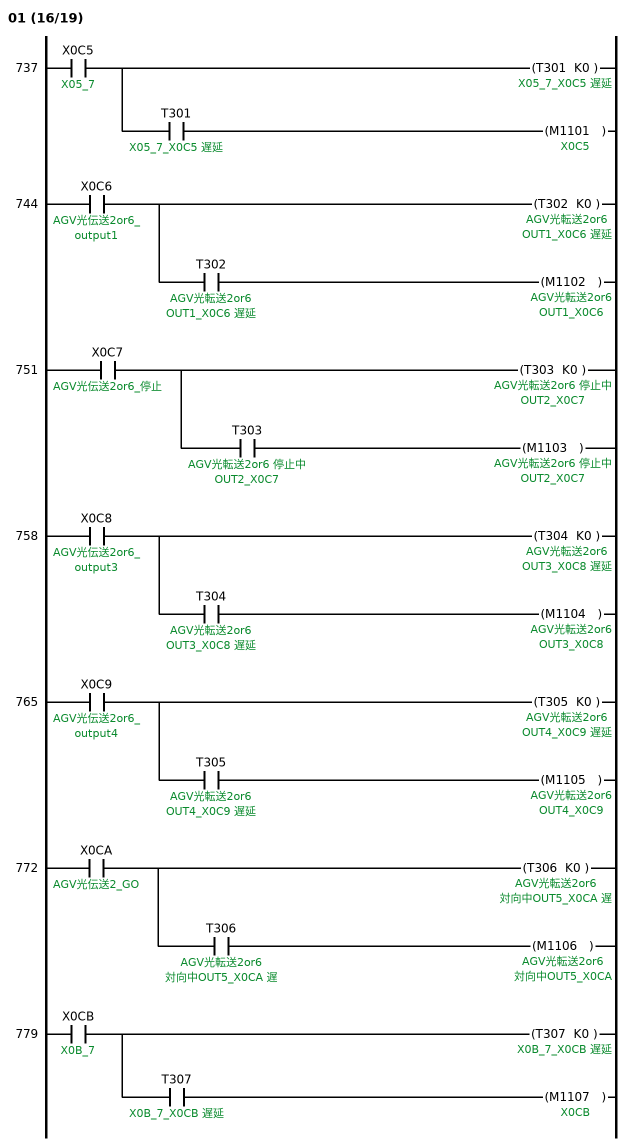
737   LD      X0C5  ; X05_7
      OUT     T301 K0  ; X05_7_X0C5 遅延
      AND     T301  ; X05_7_X0C5 遅延
      OUT     M1101  ; X0C5
744   LD      X0C6  ; AGV光伝送2or6_output1
      OUT     T302 K0  ; AGV光転送2or6 OUT1_X0C6 遅延
      AND     T302  ; AGV光転送2or6 OUT1_X0C6 遅延
      OUT     M1102  ; AGV光転送2or6 OUT1_X0C6
751   LD      X0C7  ; AGV光伝送2or6_停止
      OUT     T303 K0  ; AGV光転送2or6 停止中 OUT2_X0C7
      AND     T303  ; AGV光転送2or6 停止中 OUT2_X0C7
      OUT     M1103  ; AGV光転送2or6 停止中 OUT2_X0C7
758   LD      X0C8  ; AGV光伝送2or6_output3
      OUT     T304 K0  ; AGV光転送2or6 OUT3_X0C8 遅延
      AND     T304  ; AGV光転送2or6 OUT3_X0C8 遅延
      OUT     M1104  ; AGV光転送2or6 OUT3_X0C8
765   LD      X0C9  ; AGV光伝送2or6_output4
      OUT     T305 K0  ; AGV光転送2or6 OUT4_X0C9 遅延
      AND     T305  ; AGV光転送2or6 OUT4_X0C9 遅延
      OUT     M1105  ; AGV光転送2or6 OUT4_X0C9
772   LD      X0CA  ; AGV光伝送2_GO
      OUT     T306 K0  ; AGV光転送2or6 対向中OUT5_X0CA 遅
      AND     T306  ; AGV光転送2or6 対向中OUT5_X0CA 遅
      OUT     M1106  ; AGV光転送2or6 対向中OUT5_X0CA
779   LD      X0CB  ; X0B_7
      OUT     T307 K0  ; X0B_7_X0CB 遅延
      AND     T307  ; X0B_7_X0CB 遅延
      OUT     M1107  ; X0CB
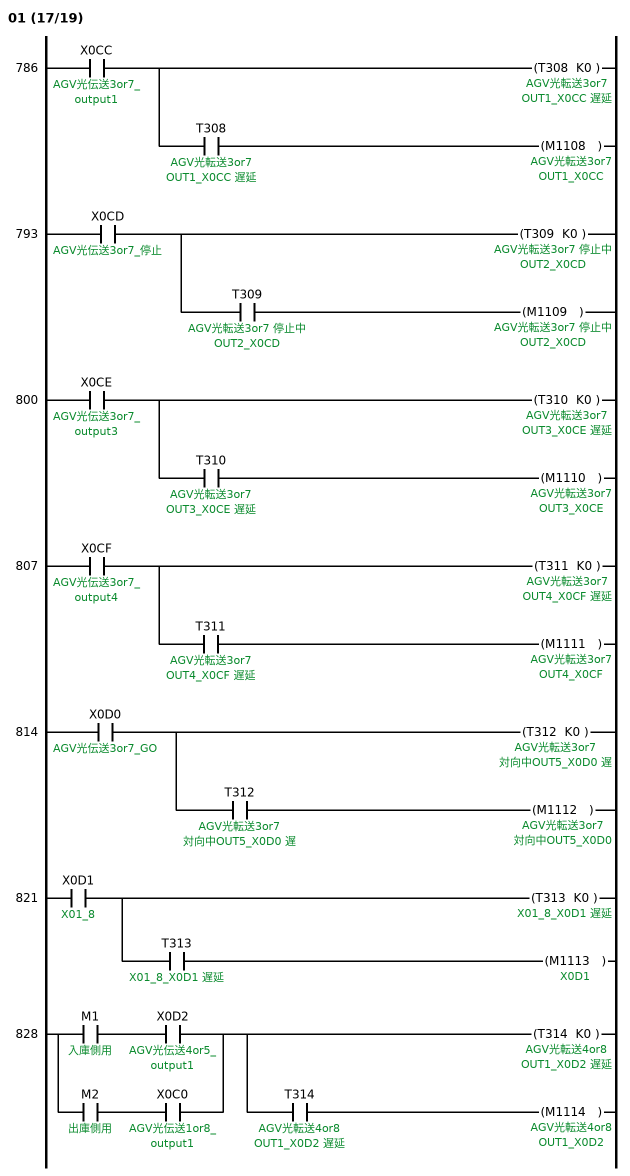
786   LD      X0CC  ; AGV光伝送3or7_output1
      OUT     T308 K0  ; AGV光転送3or7 OUT1_X0CC 遅延
      AND     T308  ; AGV光転送3or7 OUT1_X0CC 遅延
      OUT     M1108  ; AGV光転送3or7 OUT1_X0CC
793   LD      X0CD  ; AGV光伝送3or7_停止
      OUT     T309 K0  ; AGV光転送3or7 停止中 OUT2_X0CD
      AND     T309  ; AGV光転送3or7 停止中 OUT2_X0CD
      OUT     M1109  ; AGV光転送3or7 停止中 OUT2_X0CD
800   LD      X0CE  ; AGV光伝送3or7_output3
      OUT     T310 K0  ; AGV光転送3or7 OUT3_X0CE 遅延
      AND     T310  ; AGV光転送3or7 OUT3_X0CE 遅延
      OUT     M1110  ; AGV光転送3or7 OUT3_X0CE
807   LD      X0CF  ; AGV光伝送3or7_output4
      OUT     T311 K0  ; AGV光転送3or7 OUT4_X0CF 遅延
      AND     T311  ; AGV光転送3or7 OUT4_X0CF 遅延
      OUT     M1111  ; AGV光転送3or7 OUT4_X0CF
814   LD      X0D0  ; AGV光伝送3or7_GO
      OUT     T312 K0  ; AGV光転送3or7 対向中OUT5_X0D0 遅
      AND     T312  ; AGV光転送3or7 対向中OUT5_X0D0 遅
      OUT     M1112  ; AGV光転送3or7 対向中OUT5_X0D0
821   LD      X0D1  ; X01_8
      OUT     T313 K0  ; X01_8_X0D1 遅延
      AND     T313  ; X01_8_X0D1 遅延
      OUT     M1113  ; X0D1
828   LD      M1  ; 入庫側用
      AND     X0D2  ; AGV光伝送4or5_output1
      LD      M2  ; 出庫側用
      AND     X0C0  ; AGV光伝送1or8_output1
      ORB
      OUT     T314 K0  ; AGV光転送4or8 OUT1_X0D2 遅延
      AND     T314  ; AGV光転送4or8 OUT1_X0D2 遅延
      OUT     M1114  ; AGV光転送4or8 OUT1_X0D2
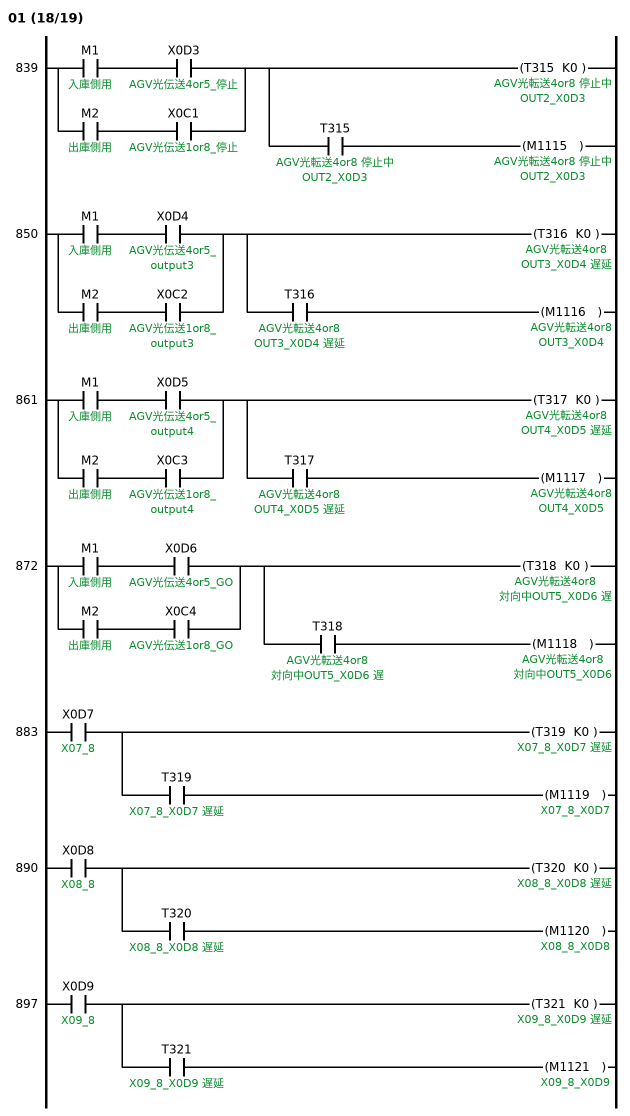
839   LD      M1  ; 入庫側用
      AND     X0D3  ; AGV光伝送4or5_停止
      LD      M2  ; 出庫側用
      AND     X0C1  ; AGV光伝送1or8_停止
      ORB
      OUT     T315 K0  ; AGV光転送4or8 停止中 OUT2_X0D3
      AND     T315  ; AGV光転送4or8 停止中 OUT2_X0D3
      OUT     M1115  ; AGV光転送4or8 停止中 OUT2_X0D3
850   LD      M1  ; 入庫側用
      AND     X0D4  ; AGV光伝送4or5_output3
      LD      M2  ; 出庫側用
      AND     X0C2  ; AGV光伝送1or8_output3
      ORB
      OUT     T316 K0  ; AGV光転送4or8 OUT3_X0D4 遅延
      AND     T316  ; AGV光転送4or8 OUT3_X0D4 遅延
      OUT     M1116  ; AGV光転送4or8 OUT3_X0D4
861   LD      M1  ; 入庫側用
      AND     X0D5  ; AGV光伝送4or5_output4
      LD      M2  ; 出庫側用
      AND     X0C3  ; AGV光伝送1or8_output4
      ORB
      OUT     T317 K0  ; AGV光転送4or8 OUT4_X0D5 遅延
      AND     T317  ; AGV光転送4or8 OUT4_X0D5 遅延
      OUT     M1117  ; AGV光転送4or8 OUT4_X0D5
872   LD      M1  ; 入庫側用
      AND     X0D6  ; AGV光伝送4or5_GO
      LD      M2  ; 出庫側用
      AND     X0C4  ; AGV光伝送1or8_GO
      ORB
      OUT     T318 K0  ; AGV光転送4or8 対向中OUT5_X0D6 遅
      AND     T318  ; AGV光転送4or8 対向中OUT5_X0D6 遅
      OUT     M1118  ; AGV光転送4or8 対向中OUT5_X0D6
883   LD      X0D7  ; X07_8
      OUT     T319 K0  ; X07_8_X0D7 遅延
      AND     T319  ; X07_8_X0D7 遅延
      OUT     M1119  ; X07_8_X0D7
890   LD      X0D8  ; X08_8
      OUT     T320 K0  ; X08_8_X0D8 遅延
      AND     T320  ; X08_8_X0D8 遅延
      OUT     M1120  ; X08_8_X0D8
897   LD      X0D9  ; X09_8
      OUT     T321 K0  ; X09_8_X0D9 遅延
      AND     T321  ; X09_8_X0D9 遅延
      OUT     M1121  ; X09_8_X0D9
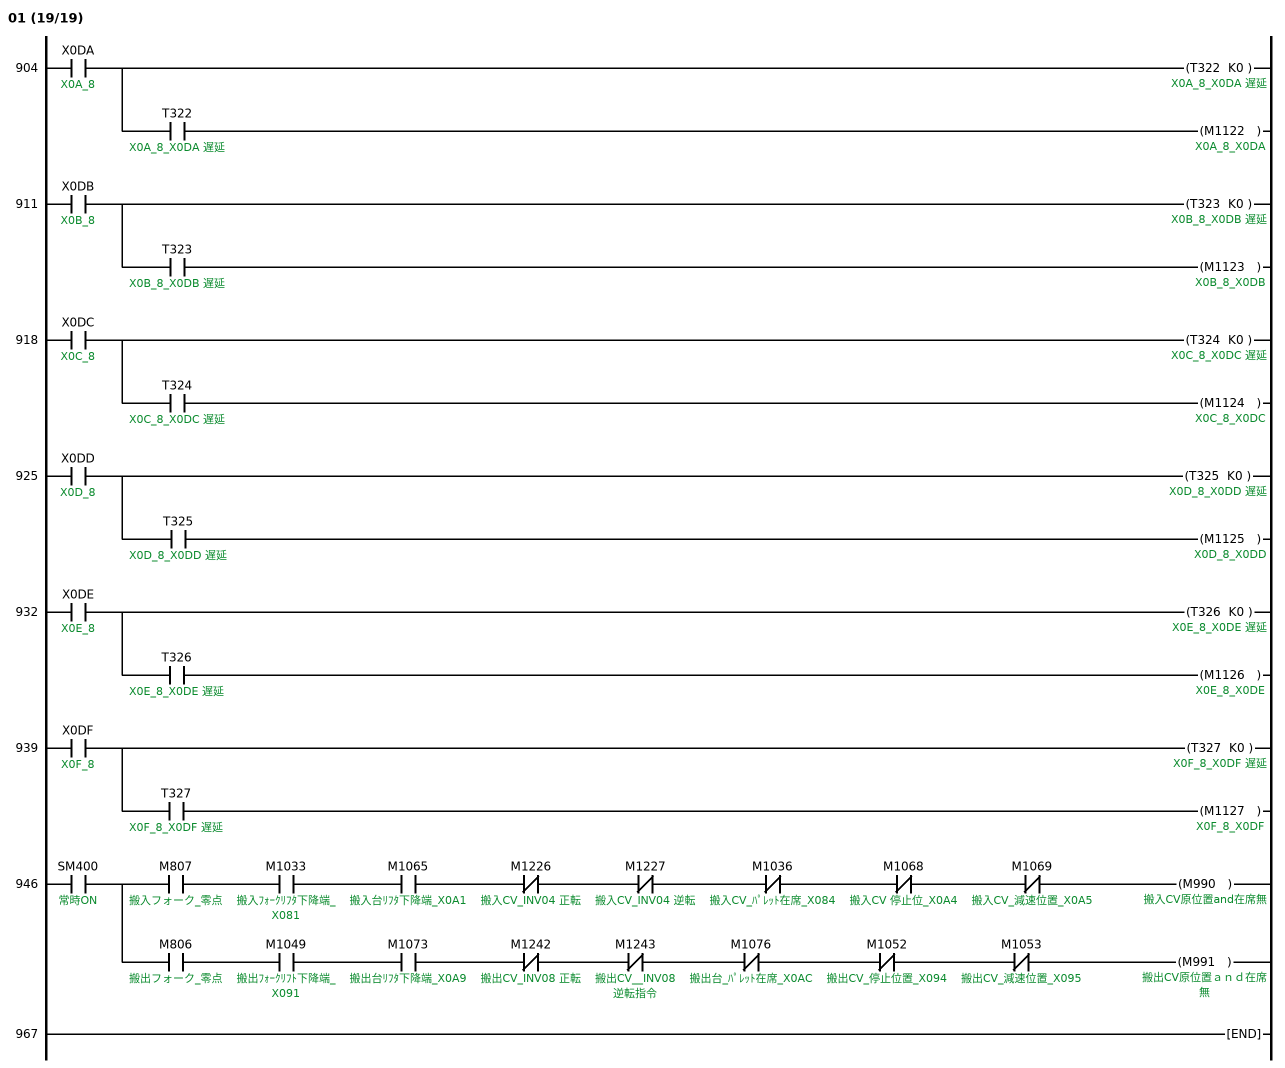
904   LD      X0DA  ; X0A_8
      OUT     T322 K0  ; X0A_8_X0DA 遅延
      AND     T322  ; X0A_8_X0DA 遅延
      OUT     M1122  ; X0A_8_X0DA
911   LD      X0DB  ; X0B_8
      OUT     T323 K0  ; X0B_8_X0DB 遅延
      AND     T323  ; X0B_8_X0DB 遅延
      OUT     M1123  ; X0B_8_X0DB
918   LD      X0DC  ; X0C_8
      OUT     T324 K0  ; X0C_8_X0DC 遅延
      AND     T324  ; X0C_8_X0DC 遅延
      OUT     M1124  ; X0C_8_X0DC
925   LD      X0DD  ; X0D_8
      OUT     T325 K0  ; X0D_8_X0DD 遅延
      AND     T325  ; X0D_8_X0DD 遅延
      OUT     M1125  ; X0D_8_X0DD
932   LD      X0DE  ; X0E_8
      OUT     T326 K0  ; X0E_8_X0DE 遅延
      AND     T326  ; X0E_8_X0DE 遅延
      OUT     M1126  ; X0E_8_X0DE
939   LD      X0DF  ; X0F_8
      OUT     T327 K0  ; X0F_8_X0DF 遅延
      AND     T327  ; X0F_8_X0DF 遅延
      OUT     M1127  ; X0F_8_X0DF
946   LD      SM400  ; 常時ON
      MPS
      AND     M807  ; 搬入フォーク_零点
      AND     M1033  ; 搬入ﾌｫｰｸﾘﾌﾀ下降端_X081
      AND     M1065  ; 搬入台ﾘﾌﾀ下降端_X0A1
      ANI     M1226  ; 搬入CV_INV04 正転
      ANI     M1227  ; 搬入CV_INV04 逆転
      ANI     M1036  ; 搬入CV_ﾊﾟﾚｯﾄ在席_X084
      ANI     M1068  ; 搬入CV 停止位_X0A4
      ANI     M1069  ; 搬入CV_減速位置_X0A5
      OUT     M990  ; 搬入CV原位置and在席無
      MPP
      AND     M806  ; 搬出フォーク_零点
      AND     M1049  ; 搬出ﾌｫｰｸﾘﾌﾄ下降端_X091
      AND     M1073  ; 搬出台ﾘﾌﾀ下降端_X0A9
      ANI     M1242  ; 搬出CV_INV08 正転
      ANI     M1243  ; 搬出CV__INV08 逆転指令
      ANI     M1076  ; 搬出台_ﾊﾟﾚｯﾄ在席_X0AC
      ANI     M1052  ; 搬出CV_停止位置_X094
      ANI     M1053  ; 搬出CV_減速位置_X095
      OUT     M991  ; 搬出CV原位置ａｎｄ在席無
967   END
END_PROGRAM

PROGRAM 02A  // CC-LinkIE XVD 入力
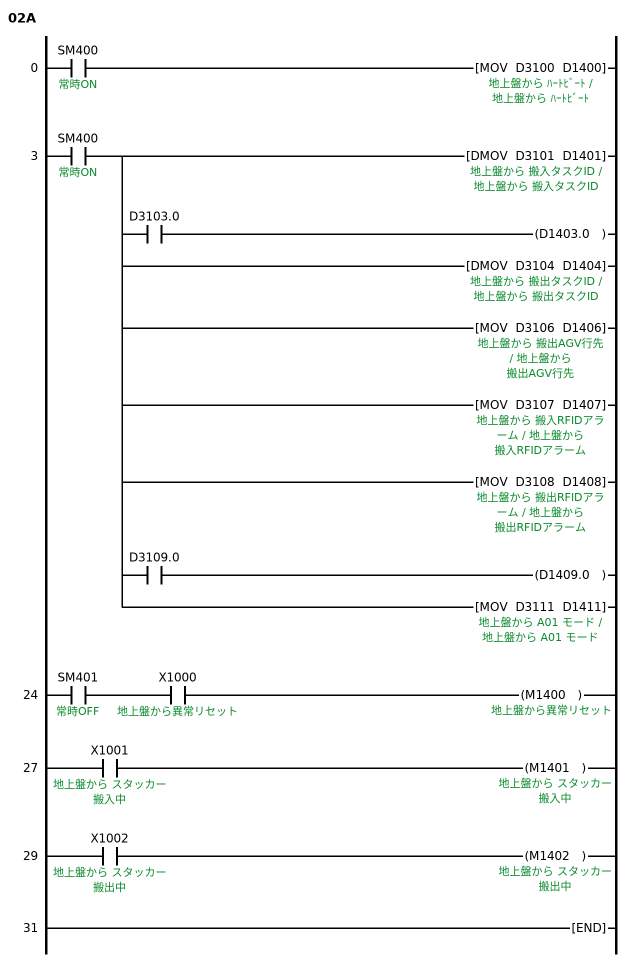
0     LD      SM400  ; 常時ON
      MOV     D3100 D1400  ; 地上盤から ﾊｰﾄﾋﾞｰﾄ / 地上盤から ﾊｰﾄﾋﾞｰﾄ
3     LD      SM400  ; 常時ON
      DMOV    D3101 D1401  ; 地上盤から 搬入タスクID / 地上盤から 搬入タスクID
      MPS
      AND     D3103.0
      OUT     D1403.0
      MPP
      DMOV    D3104 D1404  ; 地上盤から 搬出タスクID / 地上盤から 搬出タスクID
      MOV     D3106 D1406  ; 地上盤から 搬出AGV行先 / 地上盤から 搬出AGV行先
      MOV     D3107 D1407  ; 地上盤から 搬入RFIDアラーム / 地上盤から 搬入RFIDアラーム
      MOV     D3108 D1408  ; 地上盤から 搬出RFIDアラーム / 地上盤から 搬出RFIDアラーム
      MPS
      AND     D3109.0
      OUT     D1409.0
      MPP
      MOV     D3111 D1411  ; 地上盤から A01 モード / 地上盤から A01 モード
24    LD      SM401  ; 常時OFF
      AND     X1000  ; 地上盤から異常リセット
      OUT     M1400  ; 地上盤から異常リセット
27    LD      X1001  ; 地上盤から スタッカー 搬入中
      OUT     M1401  ; 地上盤から スタッカー 搬入中
29    LD      X1002  ; 地上盤から スタッカー 搬出中
      OUT     M1402  ; 地上盤から スタッカー 搬出中
31    END
END_PROGRAM

PROGRAM 05  // SAFETY
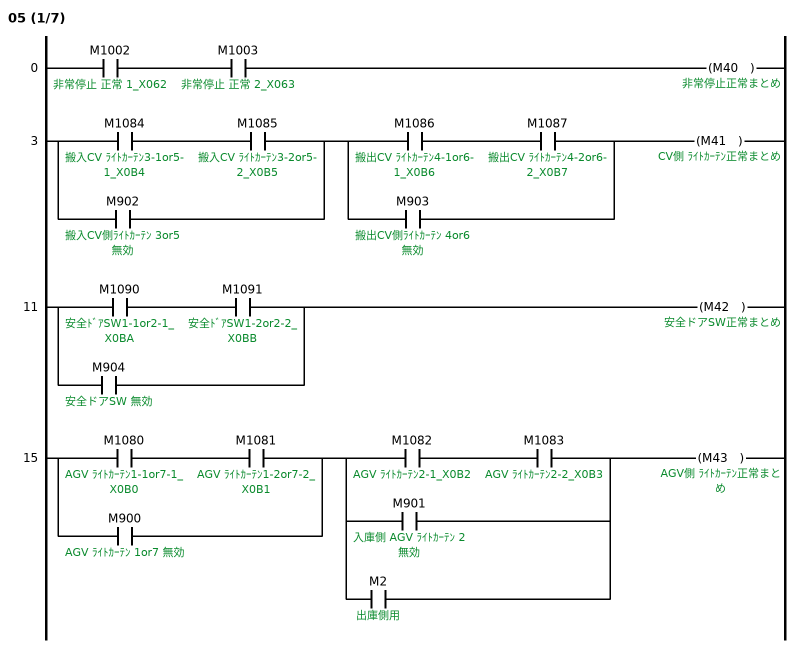
0     LD      M1002  ; 非常停止 正常 1_X062
      AND     M1003  ; 非常停止 正常 2_X063
      OUT     M40  ; 非常停止正常まとめ
3     LD      M1084  ; 搬入CV ﾗｲﾄｶｰﾃﾝ3-1or5-1_X0B4
      AND     M1085  ; 搬入CV ﾗｲﾄｶｰﾃﾝ3-2or5-2_X0B5
      OR      M902  ; 搬入CV側ﾗｲﾄｶｰﾃﾝ 3or5 無効
      LD      M1086  ; 搬出CV ﾗｲﾄｶｰﾃﾝ4-1or6-1_X0B6
      AND     M1087  ; 搬出CV ﾗｲﾄｶｰﾃﾝ4-2or6-2_X0B7
      OR      M903  ; 搬出CV側ﾗｲﾄｶｰﾃﾝ 4or6 無効
      ANB
      OUT     M41  ; CV側 ﾗｲﾄｶｰﾃﾝ正常まとめ
11    LD      M1090  ; 安全ﾄﾞｱSW1-1or2-1_X0BA
      AND     M1091  ; 安全ﾄﾞｱSW1-2or2-2_X0BB
      OR      M904  ; 安全ドアSW 無効
      OUT     M42  ; 安全ドアSW正常まとめ
15    LD      M1080  ; AGV ﾗｲﾄｶｰﾃﾝ1-1or7-1_X0B0
      AND     M1081  ; AGV ﾗｲﾄｶｰﾃﾝ1-2or7-2_X0B1
      OR      M900  ; AGV ﾗｲﾄｶｰﾃﾝ 1or7 無効
      LD      M1082  ; AGV ﾗｲﾄｶｰﾃﾝ2-1_X0B2
      AND     M1083  ; AGV ﾗｲﾄｶｰﾃﾝ2-2_X0B3
      OR      M901  ; 入庫側 AGV ﾗｲﾄｶｰﾃﾝ 2 無効
      OR      M2  ; 出庫側用
      ANB
      OUT     M43  ; AGV側 ﾗｲﾄｶｰﾃﾝ正常まとめ
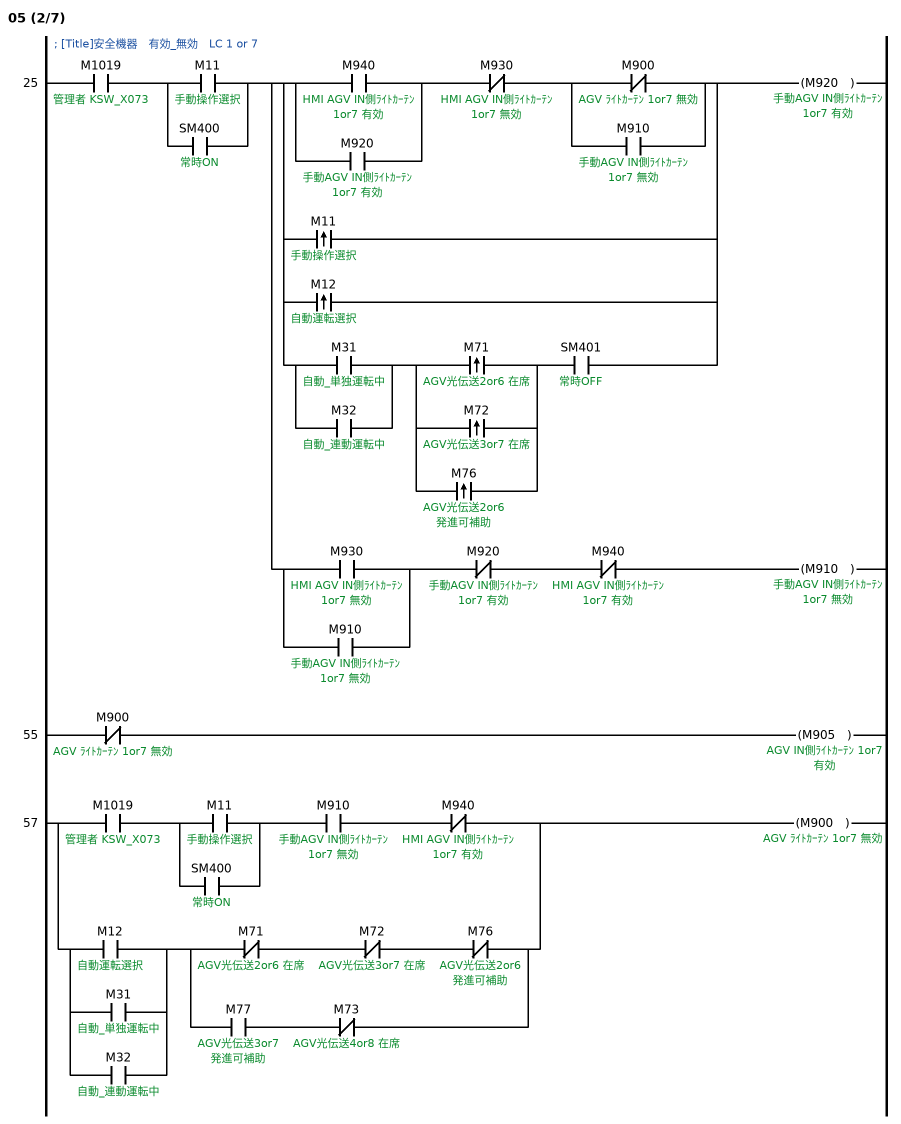
; [Title]安全機器　有効_無効　LC 1 or 7
25    LD      M1019  ; 管理者 KSW_X073
      LD      M11  ; 手動操作選択
      OR      SM400  ; 常時ON
      ANB
      MPS
      LD      M940  ; HMI AGV IN側ﾗｲﾄｶｰﾃﾝ 1or7 有効
      OR      M920  ; 手動AGV IN側ﾗｲﾄｶｰﾃﾝ 1or7 有効
      ANI     M930  ; HMI AGV IN側ﾗｲﾄｶｰﾃﾝ 1or7 無効
      LDI     M900  ; AGV ﾗｲﾄｶｰﾃﾝ 1or7 無効
      OR      M910  ; 手動AGV IN側ﾗｲﾄｶｰﾃﾝ 1or7 無効
      ANB
      ORP     M11  ; 手動操作選択
      ORP     M12  ; 自動運転選択
      LD      M31  ; 自動_単独運転中
      OR      M32  ; 自動_連動運転中
      LDP     M71  ; AGV光伝送2or6 在席
      ORP     M72  ; AGV光伝送3or7 在席
      ORP     M76  ; AGV光伝送2or6 発進可補助
      ANB
      AND     SM401  ; 常時OFF
      ORB
      ANB
      OUT     M920  ; 手動AGV IN側ﾗｲﾄｶｰﾃﾝ 1or7 有効
      MPP
      LD      M930  ; HMI AGV IN側ﾗｲﾄｶｰﾃﾝ 1or7 無効
      OR      M910  ; 手動AGV IN側ﾗｲﾄｶｰﾃﾝ 1or7 無効
      ANB
      ANI     M920  ; 手動AGV IN側ﾗｲﾄｶｰﾃﾝ 1or7 有効
      ANI     M940  ; HMI AGV IN側ﾗｲﾄｶｰﾃﾝ 1or7 有効
      OUT     M910  ; 手動AGV IN側ﾗｲﾄｶｰﾃﾝ 1or7 無効
55    LDI     M900  ; AGV ﾗｲﾄｶｰﾃﾝ 1or7 無効
      OUT     M905  ; AGV IN側ﾗｲﾄｶｰﾃﾝ 1or7 有効
57    LD      M1019  ; 管理者 KSW_X073
      LD      M11  ; 手動操作選択
      OR      SM400  ; 常時ON
      ANB
      AND     M910  ; 手動AGV IN側ﾗｲﾄｶｰﾃﾝ 1or7 無効
      ANI     M940  ; HMI AGV IN側ﾗｲﾄｶｰﾃﾝ 1or7 有効
      LD      M12  ; 自動運転選択
      OR      M31  ; 自動_単独運転中
      OR      M32  ; 自動_連動運転中
      LDI     M71  ; AGV光伝送2or6 在席
      ANI     M72  ; AGV光伝送3or7 在席
      ANI     M76  ; AGV光伝送2or6 発進可補助
      LD      M77  ; AGV光伝送3or7 発進可補助
      ANI     M73  ; AGV光伝送4or8 在席
      ORB
      ANB
      ORB
      OUT     M900  ; AGV ﾗｲﾄｶｰﾃﾝ 1or7 無効
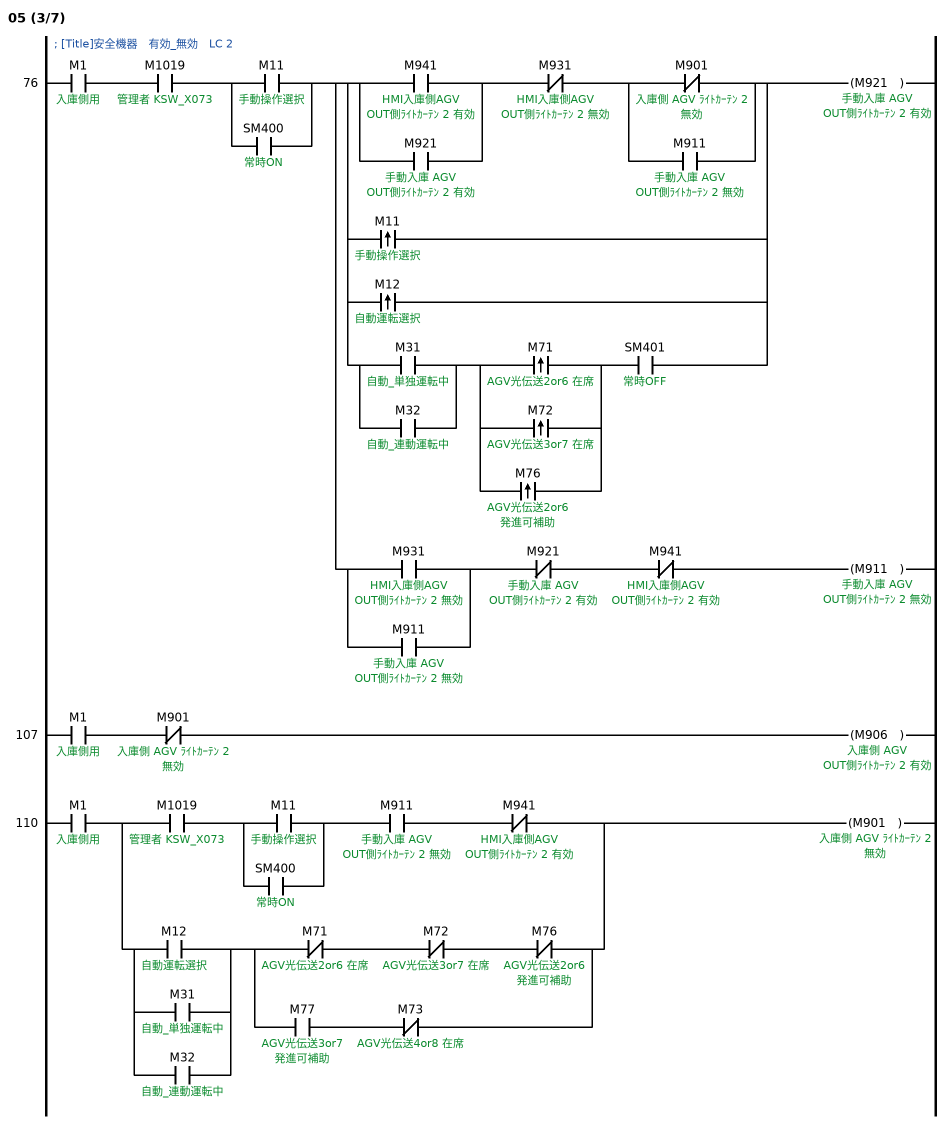
; [Title]安全機器　有効_無効　LC 2
76    LD      M1  ; 入庫側用
      AND     M1019  ; 管理者 KSW_X073
      LD      M11  ; 手動操作選択
      OR      SM400  ; 常時ON
      ANB
      MPS
      LD      M941  ; HMI入庫側AGV OUT側ﾗｲﾄｶｰﾃﾝ 2 有効
      OR      M921  ; 手動入庫 AGV OUT側ﾗｲﾄｶｰﾃﾝ 2 有効
      ANI     M931  ; HMI入庫側AGV OUT側ﾗｲﾄｶｰﾃﾝ 2 無効
      LDI     M901  ; 入庫側 AGV ﾗｲﾄｶｰﾃﾝ 2 無効
      OR      M911  ; 手動入庫 AGV OUT側ﾗｲﾄｶｰﾃﾝ 2 無効
      ANB
      ORP     M11  ; 手動操作選択
      ORP     M12  ; 自動運転選択
      LD      M31  ; 自動_単独運転中
      OR      M32  ; 自動_連動運転中
      LDP     M71  ; AGV光伝送2or6 在席
      ORP     M72  ; AGV光伝送3or7 在席
      ORP     M76  ; AGV光伝送2or6 発進可補助
      ANB
      AND     SM401  ; 常時OFF
      ORB
      ANB
      OUT     M921  ; 手動入庫 AGV OUT側ﾗｲﾄｶｰﾃﾝ 2 有効
      MPP
      LD      M931  ; HMI入庫側AGV OUT側ﾗｲﾄｶｰﾃﾝ 2 無効
      OR      M911  ; 手動入庫 AGV OUT側ﾗｲﾄｶｰﾃﾝ 2 無効
      ANB
      ANI     M921  ; 手動入庫 AGV OUT側ﾗｲﾄｶｰﾃﾝ 2 有効
      ANI     M941  ; HMI入庫側AGV OUT側ﾗｲﾄｶｰﾃﾝ 2 有効
      OUT     M911  ; 手動入庫 AGV OUT側ﾗｲﾄｶｰﾃﾝ 2 無効
107   LD      M1  ; 入庫側用
      ANI     M901  ; 入庫側 AGV ﾗｲﾄｶｰﾃﾝ 2 無効
      OUT     M906  ; 入庫側 AGV OUT側ﾗｲﾄｶｰﾃﾝ 2 有効
110   LD      M1  ; 入庫側用
      LD      M1019  ; 管理者 KSW_X073
      LD      M11  ; 手動操作選択
      OR      SM400  ; 常時ON
      ANB
      AND     M911  ; 手動入庫 AGV OUT側ﾗｲﾄｶｰﾃﾝ 2 無効
      ANI     M941  ; HMI入庫側AGV OUT側ﾗｲﾄｶｰﾃﾝ 2 有効
      LD      M12  ; 自動運転選択
      OR      M31  ; 自動_単独運転中
      OR      M32  ; 自動_連動運転中
      LDI     M71  ; AGV光伝送2or6 在席
      ANI     M72  ; AGV光伝送3or7 在席
      ANI     M76  ; AGV光伝送2or6 発進可補助
      LD      M77  ; AGV光伝送3or7 発進可補助
      ANI     M73  ; AGV光伝送4or8 在席
      ORB
      ANB
      ORB
      ANB
      OUT     M901  ; 入庫側 AGV ﾗｲﾄｶｰﾃﾝ 2 無効
